LIN {X 0,Y 354.821,Z 300.916,A -85,B 0,C 180,E1 -13284.301,E2 -13284.301} C_VEL
LIN {X 0,Y 354.785,Z 300.918,A -85,B 0,C 180,E1 -13287.666,E2 -13287.666} C_VEL
LIN {X 0,Y 354.8,Z 300.915,A -85,B 0,C 180,E1 -13291.614,E2 -13291.614} C_VEL
LIN {X 0,Y 354.849,Z 300.908,A -85,B 0,C 180,E1 -13295.423,E2 -13295.423} C_VEL
LIN {X 0,Y 354.825,Z 300.912,A -85,B 0,C 180,E1 -13299.113,E2 -13299.113} C_VEL
LIN {X 0,Y 354.896,Z 300.903,A -85,B 0,C 180,E1 -13302.72,E2 -13302.72} C_VEL
LIN {X 0,Y 354.949,Z 300.895,A -85,B 0,C 180,E1 -13306.255,E2 -13306.255} C_VEL
LIN {X 0,Y 354.954,Z 300.896,A -85,B 0,C 180,E1 -13309.735,E2 -13309.735} C_VEL
LIN {X 0,Y 355.087,Z 300.878,A -85,B 0,C 180,E1 -13313.18,E2 -13313.18} C_VEL
LIN {X 0,Y 355.243,Z 300.859,A -85,B 0,C 180,E1 -13317.732,E2 -13317.732} C_VEL
LIN {X 0,Y 355.33,Z 300.85,A -85,B 0,C 180,E1 -13320,E2 -13320} C_VEL
LIN {X 0,Y 355.243,Z 300.859,A -85,B 0,C 180,E1 -13322.268,E2 -13322.268} C_VEL
LIN {X 0,Y 355.087,Z 300.878,A -85,B 0,C 180,E1 -13326.82,E2 -13326.82} C_VEL
LIN {X 0,Y 354.954,Z 300.896,A -85,B 0,C 180,E1 -13330.265,E2 -13330.265} C_VEL
LIN {X 0,Y 354.94,Z 300.899,A -85,B 0,C 180,E1 -13334.019,E2 -13334.019} C_VEL
LIN {X 0,Y 354.92,Z 300.901,A -85,B 0,C 180,E1 -13338.108,E2 -13338.108} C_VEL
LIN {X 0,Y 354.814,Z 300.913,A -85,B 0,C 180,E1 -13342.107,E2 -13342.107} C_VEL
LIN {X 0,Y 354.896,Z 300.904,A -85,B 0,C 180,E1 -13345.828,E2 -13345.828} C_VEL
LIN {X 0,Y 354.816,Z 300.917,A -85,B 0,C 180,E1 -13349.682,E2 -13349.682} C_VEL
LIN {X 0,Y 354.804,Z 300.923,A -85,B 0,C 180,E1 -13353.702,E2 -13353.702} C_VEL
LIN {X 0,Y 354.795,Z 300.924,A -85,B 0,C 180,E1 -13356.46,E2 -13356.46} C_VEL
LIN {X 0,Y 354.823,Z 300.917,A -85,B 0,C 180,E1 -13359.424,E2 -13359.424} C_VEL
LIN {X 0,Y 354.942,Z 301.94,A -85,B 0,C 180,E1 -13361.2,E2 -13361.2} C_VEL
LIN {X 0,Y 355.522,Z 305.414,A -85,B 0,C 180,E1 -13364.631,E2 -13364.631} C_VEL
LIN {X 0,Y 355.791,Z 308.9,A -85,B 0,C 180,E1 -13367.809,E2 -13367.809} C_VEL
LIN {X 0,Y 355.65,Z 312.374,A -85,B 0,C 180,E1 -13370.776,E2 -13370.776} C_VEL
LIN {X 0,Y 355.208,Z 316.65,A -85,B 0,C 180,E1 -13374.214,E2 -13374.214} C_VEL
LIN {X 0,Y 354.802,Z 321.128,A -85,B 0,C 180,E1 -13377.668,E2 -13377.668} C_VEL
LIN {X 0,Y 354.435,Z 325.194,A -85,B 0,C 180,E1 -13380.711,E2 -13380.711} C_VEL
LIN {X 0,Y 355.437,Z 328.521,A -85,B 0,C 180,E1 -13380.888,E2 -13380.888} C_VEL
LIN {X 0,Y 360.165,Z 342.303,A -85,B 0,C 180,E1 -13381.741,E2 -13381.741} C_VEL
LIN {X 0,Y 364.264,Z 357.145,A -85,B 0,C 180,E1 -13382.781,E2 -13382.781} C_VEL
LIN {X 0,Y 367.132,Z 370.992,A -85,B 0,C 180,E1 -13383.878,E2 -13383.878} C_VEL
LIN {X 0,Y 367.5,Z 375.118,A -85,B 0,C 180,E1 -13384.21,E2 -13384.21} C_VEL
LIN {X 0,Y 365.724,Z 389.395,A -85,B 0,C 180,E1 -13385.294,E2 -13385.294} C_VEL
LIN {X 0,Y 363.918,Z 402.392,A -85,B 0,C 180,E1 -13386.527,E2 -13386.527} C_VEL
LIN {X 0,Y 362.123,Z 414.391,A -85,B 0,C 180,E1 -13387.912,E2 -13387.912} C_VEL
LIN {X 0,Y 360.283,Z 425.503,A -85,B 0,C 180,E1 -13389.444,E2 -13389.444} C_VEL
LIN {X 0,Y 358.7,Z 435.728,A -85,B 0,C 180,E1 -13391.138,E2 -13391.138} C_VEL
LIN {X 0,Y 357.065,Z 445.72,A -85,B 0,C 180,E1 -13393.123,E2 -13393.123} C_VEL
LIN {X 0,Y 355.76,Z 454.016,A -85,B 0,C 180,E1 -13395.119,E2 -13395.119} C_VEL
LIN {X 0,Y 354.77,Z 461.81,A -85,B 0,C 180,E1 -13397.413,E2 -13397.413} C_VEL
LIN {X 0,Y 353.938,Z 468.009,A -85,B 0,C 180,E1 -13399.705,E2 -13399.705} C_VEL
LIN {X 0,Y 353.512,Z 472.803,A -85,B 0,C 180,E1 -13402,E2 -13402} C_VEL
LIN {X 0,Y 353.26,Z 476.314,A -85,B 0,C 180,E1 -13404.291,E2 -13404.291} C_VEL
LIN {X 0,Y 353.182,Z 478.624,A -85,B 0,C 180,E1 -13406.577,E2 -13406.577} C_VEL
LIN {X 0,Y 353.144,Z 479.785,A -85,B 0,C 180,E1 -13408.859,E2 -13408.859} C_VEL
LIN {X 0,Y 353.144,Z 479.783,A -85,B 0,C 180,E1 -13411.14,E2 -13411.14} C_VEL
LIN {X 0,Y 353.183,Z 478.613,A -85,B 0,C 180,E1 -13413.422,E2 -13413.422} C_VEL
LIN {X 0,Y 353.312,Z 475.97,A -85,B 0,C 180,E1 -13415.965,E2 -13415.965} C_VEL
LIN {X 0,Y 353.601,Z 471.718,A -85,B 0,C 180,E1 -13418.572,E2 -13418.572} C_VEL
LIN {X 0,Y 354.061,Z 466.558,A -85,B 0,C 180,E1 -13420.869,E2 -13420.869} C_VEL
LIN {X 0,Y 354.957,Z 459.959,A -85,B 0,C 180,E1 -13423.161,E2 -13423.161} C_VEL
LIN {X 0,Y 355.943,Z 452.851,A -85,B 0,C 180,E1 -13425.165,E2 -13425.165} C_VEL
LIN {X 0,Y 357.256,Z 444.313,A -85,B 0,C 180,E1 -13427.162,E2 -13427.162} C_VEL
LIN {X 0,Y 358.709,Z 435.666,A -85,B 0,C 180,E1 -13428.86,E2 -13428.86} C_VEL
LIN {X 0,Y 360.406,Z 425.069,A -85,B 0,C 180,E1 -13430.608,E2 -13430.608} C_VEL
LIN {X 0,Y 362.266,Z 413.241,A -85,B 0,C 180,E1 -13432.228,E2 -13432.228} C_VEL
LIN {X 0,Y 364.288,Z 399.662,A -85,B 0,C 180,E1 -13433.748,E2 -13433.748} C_VEL
LIN {X 0,Y 366.179,Z 386.045,A -85,B 0,C 180,E1 -13434.975,E2 -13434.975} C_VEL
LIN {X 0,Y 367.506,Z 374.442,A -85,B 0,C 180,E1 -13435.827,E2 -13435.827} C_VEL
LIN {X 0,Y 365.476,Z 363.038,A -85,B 0,C 180,E1 -13436.76,E2 -13436.76} C_VEL
LIN {X 0,Y 362.281,Z 349.698,A -85,B 0,C 180,E1 -13437.747,E2 -13437.747} C_VEL
LIN {X 0,Y 357.545,Z 334.313,A -85,B 0,C 180,E1 -13438.751,E2 -13438.751} C_VEL
LIN {X 0,Y 354.548,Z 326.07,A -85,B 0,C 180,E1 -13439.238,E2 -13439.238} C_VEL
LIN {X 0,Y 354.421,Z 325.198,A -85,B 0,C 180,E1 -13439.285,E2 -13439.285} C_VEL
LIN {X 0,Y 354.8,Z 321.14,A -85,B 0,C 180,E1 -13442.331,E2 -13442.331} C_VEL
LIN {X 0,Y 355.205,Z 316.687,A -85,B 0,C 180,E1 -13445.785,E2 -13445.785} C_VEL
LIN {X 0,Y 355.651,Z 312.432,A -85,B 0,C 180,E1 -13449.222,E2 -13449.222} C_VEL
LIN {X 0,Y 355.788,Z 308.925,A -85,B 0,C 180,E1 -13452.19,E2 -13452.19} C_VEL
LIN {X 0,Y 355.521,Z 305.416,A -85,B 0,C 180,E1 -13455.368,E2 -13455.368} C_VEL
LIN {X 0,Y 354.878,Z 301.531,A -85,B 0,C 180,E1 -13459.192,E2 -13459.192} C_VEL
LIN {X 0,Y 354.81,Z 300.916,A -85,B 0,C 180,E1 -13460.665,E2 -13460.665} C_VEL
LIN {X 0,Y 354.815,Z 300.917,A -85,B 0,C 180,E1 -13464.3,E2 -13464.3} C_VEL
LIN {X 0,Y 354.78,Z 300.924,A -85,B 0,C 180,E1 -13467.666,E2 -13467.666} C_VEL
LIN {X 0,Y 354.84,Z 300.914,A -85,B 0,C 180,E1 -13471.618,E2 -13471.618} C_VEL
LIN {X 0,Y 354.892,Z 300.905,A -85,B 0,C 180,E1 -13474.172,E2 -13474.172} C_VEL
LIN {X 0,Y 354.827,Z 300.911,A -85,B 0,C 180,E1 -13477.894,E2 -13477.894} C_VEL
LIN {X 0,Y 354.916,Z 300.9,A -85,B 0,C 180,E1 -13481.891,E2 -13481.891} C_VEL
LIN {X 0,Y 354.935,Z 300.897,A -85,B 0,C 180,E1 -13485.981,E2 -13485.981} C_VEL
LIN {X 0,Y 354.949,Z 300.896,A -85,B 0,C 180,E1 -13489.735,E2 -13489.735} C_VEL
LIN {X 0,Y 355.082,Z 300.879,A -85,B 0,C 180,E1 -13493.18,E2 -13493.18} C_VEL
LIN {X 0,Y 355.239,Z 300.855,A -85,B 0,C 180,E1 -13497.732,E2 -13497.732} C_VEL
LIN {X 0,Y 355.345,Z 300.849,A -85,B 0,C 180,E1 -13500,E2 -13500} C_VEL
LIN {X 0,Y 355.239,Z 300.859,A -85,B 0,C 180,E1 -13502.268,E2 -13502.268} C_VEL
LIN {X 0,Y 355.082,Z 300.879,A -85,B 0,C 180,E1 -13506.82,E2 -13506.82} C_VEL
LIN {X 0,Y 354.949,Z 300.897,A -85,B 0,C 180,E1 -13510.265,E2 -13510.265} C_VEL
LIN {X 0,Y 354.935,Z 300.897,A -85,B 0,C 180,E1 -13514.019,E2 -13514.019} C_VEL
LIN {X 0,Y 354.916,Z 300.898,A -85,B 0,C 180,E1 -13518.109,E2 -13518.109} C_VEL
LIN {X 0,Y 354.829,Z 300.911,A -85,B 0,C 180,E1 -13522.107,E2 -13522.107} C_VEL
LIN {X 0,Y 354.893,Z 300.904,A -85,B 0,C 180,E1 -13525.828,E2 -13525.828} C_VEL
LIN {X 0,Y 354.812,Z 300.91,A -85,B 0,C 180,E1 -13529.683,E2 -13529.683} C_VEL
LIN {X 0,Y 354.801,Z 300.913,A -85,B 0,C 180,E1 -13533.703,E2 -13533.703} C_VEL
LIN {X 0,Y 354.793,Z 300.915,A -85,B 0,C 180,E1 -13536.46,E2 -13536.46} C_VEL
LIN {X 0,Y 354.819,Z 300.914,A -85,B 0,C 180,E1 -13539.424,E2 -13539.424} C_VEL
LIN {X 0,Y 354.785,Z 300.92,A -85,B 0,C 180,E1 -13542.868,E2 -13542.868} C_VEL
LIN {X 0,Y 355.185,Z 303.837,A -85,B 0,C 180,E1 -13546.17,E2 -13546.17} C_VEL
LIN {X 0,Y 355.333,Z 306.315,A -85,B 0,C 180,E1 -13548.728,E2 -13548.728} C_VEL
LIN {X 0,Y 355.07,Z 309.877,A -85,B 0,C 180,E1 -13552.152,E2 -13552.152} C_VEL
LIN {X 0,Y 354.85,Z 312.922,A -85,B 0,C 180,E1 -13554.946,E2 -13554.946} C_VEL
LIN {X 0,Y 354.487,Z 317.485,A -85,B 0,C 180,E1 -13558.972,E2 -13558.972} C_VEL
LIN {X 0,Y 354.323,Z 319.729,A -85,B 0,C 180,E1 -13560.779,E2 -13560.779} C_VEL
LIN {X 0,Y 355.465,Z 323.077,A -85,B 0,C 180,E1 -13560.969,E2 -13560.969} C_VEL
LIN {X 0,Y 360.81,Z 337.991,A -85,B 0,C 180,E1 -13561.937,E2 -13561.937} C_VEL
LIN {X 0,Y 364.609,Z 351.156,A -85,B 0,C 180,E1 -13562.885,E2 -13562.885} C_VEL
LIN {X 0,Y 367.818,Z 365.813,A -85,B 0,C 180,E1 -13564.074,E2 -13564.074} C_VEL
LIN {X 0,Y 366.527,Z 379.062,A -85,B 0,C 180,E1 -13565.05,E2 -13565.05} C_VEL
LIN {X 0,Y 364.645,Z 392.749,A -85,B 0,C 180,E1 -13566.277,E2 -13566.277} C_VEL
LIN {X 0,Y 362.816,Z 405.219,A -85,B 0,C 180,E1 -13567.658,E2 -13567.658} C_VEL
LIN {X 0,Y 361.193,Z 415.771,A -85,B 0,C 180,E1 -13569.063,E2 -13569.063} C_VEL
LIN {X 0,Y 359.307,Z 427.192,A -85,B 0,C 180,E1 -13570.876,E2 -13570.876} C_VEL
LIN {X 0,Y 357.628,Z 437.465,A -85,B 0,C 180,E1 -13572.857,E2 -13572.857} C_VEL
LIN {X 0,Y 356.265,Z 445.996,A -85,B 0,C 180,E1 -13574.849,E2 -13574.849} C_VEL
LIN {X 0,Y 355.264,Z 453.095,A -85,B 0,C 180,E1 -13576.851,E2 -13576.851} C_VEL
LIN {X 0,Y 354.278,Z 459.684,A -85,B 0,C 180,E1 -13579.138,E2 -13579.138} C_VEL
LIN {X 0,Y 353.749,Z 464.834,A -85,B 0,C 180,E1 -13581.431,E2 -13581.431} C_VEL
LIN {X 0,Y 353.443,Z 468.827,A -85,B 0,C 180,E1 -13583.837,E2 -13583.837} C_VEL
LIN {X 0,Y 353.284,Z 470.71,A -85,B 0,C 180,E1 -13585.436,E2 -13585.436} C_VEL
LIN {X 0,Y 353.167,Z 472.459,A -85,B 0,C 180,E1 -13587.72,E2 -13587.72} C_VEL
LIN {X 0,Y 353.174,Z 473.069,A -85,B 0,C 180,E1 -13590,E2 -13590} C_VEL
LIN {X 0,Y 353.167,Z 472.503,A -85,B 0,C 180,E1 -13592.281,E2 -13592.281} C_VEL
LIN {X 0,Y 353.282,Z 470.812,A -85,B 0,C 180,E1 -13594.564,E2 -13594.564} C_VEL
LIN {X 0,Y 353.428,Z 467.96,A -85,B 0,C 180,E1 -13596.853,E2 -13596.853} C_VEL
LIN {X 0,Y 353.841,Z 463.877,A -85,B 0,C 180,E1 -13599.143,E2 -13599.143} C_VEL
LIN {X 0,Y 354.441,Z 458.466,A -85,B 0,C 180,E1 -13601.437,E2 -13601.437} C_VEL
LIN {X 0,Y 355.227,Z 453.413,A -85,B 0,C 180,E1 -13603.151,E2 -13603.151} C_VEL
LIN {X 0,Y 356.17,Z 446.386,A -85,B 0,C 180,E1 -13605.156,E2 -13605.156} C_VEL
LIN {X 0,Y 357.56,Z 437.93,A -85,B 0,C 180,E1 -13607.148,E2 -13607.148} C_VEL
LIN {X 0,Y 359.238,Z 427.749,A -85,B 0,C 180,E1 -13609.129,E2 -13609.129} C_VEL
LIN {X 0,Y 360.999,Z 417.043,A -85,B 0,C 180,E1 -13610.856,E2 -13610.856} C_VEL
LIN {X 0,Y 362.878,Z 404.837,A -85,B 0,C 180,E1 -13612.489,E2 -13612.489} C_VEL
LIN {X 0,Y 364.729,Z 392.289,A -85,B 0,C 180,E1 -13613.869,E2 -13613.869} C_VEL
LIN {X 0,Y 366.575,Z 379.12,A -85,B 0,C 180,E1 -13615.046,E2 -13615.046} C_VEL
LIN {X 0,Y 367.907,Z 366.961,A -85,B 0,C 180,E1 -13615.936,E2 -13615.936} C_VEL
LIN {X 0,Y 366.464,Z 359.08,A -85,B 0,C 180,E1 -13616.593,E2 -13616.593} C_VEL
LIN {X 0,Y 362.78,Z 344.309,A -85,B 0,C 180,E1 -13617.722,E2 -13617.722} C_VEL
LIN {X 0,Y 357.834,Z 329.329,A -85,B 0,C 180,E1 -13618.749,E2 -13618.749} C_VEL
LIN {X 0,Y 354.379,Z 320.072,A -85,B 0,C 180,E1 -13619.316,E2 -13619.316} C_VEL
LIN {X 0,Y 354.31,Z 319.565,A -85,B 0,C 180,E1 -13619.375,E2 -13619.375} C_VEL
LIN {X 0,Y 354.393,Z 318.435,A -85,B 0,C 180,E1 -13620.347,E2 -13620.347} C_VEL
LIN {X 0,Y 353.819,Z 317.434,A -85,B 0,C 180,E1 -13621.284,E2 -13621.284} C_VEL
LIN {X 0,Y 351.083,Z 316.043,A -85,B 0,C 180,E1 -13622.816,E2 -13622.816} C_VEL
LIN {X 0,Y 348.77,Z 314.97,A -85,B 0,C 180,E1 -13624.058,E2 -13624.058} C_VEL
LIN {X 0,Y 347.843,Z 314.059,A -85,B 0,C 180,E1 -13625.014,E2 -13625.014} C_VEL
LIN {X 0,Y 347.804,Z 313.72,A -85,B 0,C 180,E1 -13625.336,E2 -13625.336} C_VEL
LIN {X 0,Y 348.101,Z 310.13,A -85,B 0,C 180,E1 -13628.746,E2 -13628.746} C_VEL
LIN {X 0,Y 348.326,Z 307.061,A -85,B 0,C 180,E1 -13631.745,E2 -13631.745} C_VEL
LIN {X 0,Y 348.084,Z 304.026,A -85,B 0,C 180,E1 -13634.964,E2 -13634.964} C_VEL
LIN {X 0,Y 347.856,Z 302.5,A -85,B 0,C 180,E1 -13636.663,E2 -13636.663} C_VEL
LIN {X 0,Y 347.75,Z 301.794,A -85,B 0,C 180,E1 -13638.397,E2 -13638.397} C_VEL
LIN {X 0,Y 347.773,Z 301.793,A -85,B 0,C 180,E1 -13642.011,E2 -13642.011} C_VEL
LIN {X 0,Y 347.743,Z 301.797,A -85,B 0,C 180,E1 -13645.536,E2 -13645.536} C_VEL
LIN {X 0,Y 347.744,Z 301.796,A -85,B 0,C 180,E1 -13648.3,E2 -13648.3} C_VEL
LIN {X 0,Y 347.745,Z 301.794,A -85,B 0,C 180,E1 -13650.984,E2 -13650.984} C_VEL
LIN {X 0,Y 347.753,Z 301.791,A -85,B 0,C 180,E1 -13653.601,E2 -13653.601} C_VEL
LIN {X 0,Y 347.768,Z 301.791,A -85,B 0,C 180,E1 -13656.16,E2 -13656.16} C_VEL
LIN {X 0,Y 347.81,Z 301.787,A -85,B 0,C 180,E1 -13659.909,E2 -13659.909} C_VEL
LIN {X 0,Y 347.865,Z 301.779,A -85,B 0,C 180,E1 -13662.359,E2 -13662.359} C_VEL
LIN {X 0,Y 347.896,Z 301.776,A -85,B 0,C 180,E1 -13665.971,E2 -13665.971} C_VEL
LIN {X 0,Y 347.894,Z 301.776,A -85,B 0,C 180,E1 -13669.524,E2 -13669.524} C_VEL
LIN {X 0,Y 348.054,Z 301.755,A -85,B 0,C 180,E1 -13673.041,E2 -13673.041} C_VEL
LIN {X 0,Y 348.206,Z 301.735,A -85,B 0,C 180,E1 -13677.686,E2 -13677.686} C_VEL
LIN {X 0,Y 348.281,Z 301.728,A -85,B 0,C 180,E1 -13680,E2 -13680} C_VEL
LIN {X 0,Y 348.206,Z 301.736,A -85,B 0,C 180,E1 -13682.313,E2 -13682.313} C_VEL
LIN {X 0,Y 348.053,Z 301.754,A -85,B 0,C 180,E1 -13686.959,E2 -13686.959} C_VEL
LIN {X 0,Y 347.894,Z 301.777,A -85,B 0,C 180,E1 -13690.475,E2 -13690.475} C_VEL
LIN {X 0,Y 347.896,Z 301.776,A -85,B 0,C 180,E1 -13694.15,E2 -13694.15} C_VEL
LIN {X 0,Y 347.889,Z 301.778,A -85,B 0,C 180,E1 -13698.29,E2 -13698.29} C_VEL
LIN {X 0,Y 347.766,Z 301.793,A -85,B 0,C 180,E1 -13701.626,E2 -13701.626} C_VEL
LIN {X 0,Y 347.809,Z 301.785,A -85,B 0,C 180,E1 -13705.109,E2 -13705.109} C_VEL
LIN {X 0,Y 347.806,Z 301.789,A -85,B 0,C 180,E1 -13707.694,E2 -13707.694} C_VEL
LIN {X 0,Y 347.747,Z 301.799,A -85,B 0,C 180,E1 -13710.348,E2 -13710.348} C_VEL
LIN {X 0,Y 347.746,Z 301.802,A -85,B 0,C 180,E1 -13714.044,E2 -13714.044} C_VEL
LIN {X 0,Y 347.759,Z 301.8,A -85,B 0,C 180,E1 -13717.321,E2 -13717.321} C_VEL
LIN {X 0,Y 347.763,Z 301.892,A -85,B 0,C 180,E1 -13719.83,E2 -13719.83} C_VEL
LIN {X 0,Y 348.307,Z 305.371,A -85,B 0,C 180,E1 -13723.415,E2 -13723.415} C_VEL
LIN {X 0,Y 348.728,Z 308.572,A -85,B 0,C 180,E1 -13726.512,E2 -13726.512} C_VEL
LIN {X 0,Y 348.767,Z 310.573,A -85,B 0,C 180,E1 -13728.319,E2 -13728.319} C_VEL
LIN {X 0,Y 348.529,Z 314.056,A -85,B 0,C 180,E1 -13731.31,E2 -13731.31} C_VEL
LIN {X 0,Y 348.172,Z 317.564,A -85,B 0,C 180,E1 -13734.171,E2 -13734.171} C_VEL
LIN {X 0,Y 347.819,Z 321.054,A -85,B 0,C 180,E1 -13736.937,E2 -13736.937} C_VEL
LIN {X 0,Y 347.447,Z 325.114,A -85,B 0,C 180,E1 -13740.055,E2 -13740.055} C_VEL
LIN {X 0,Y 348.341,Z 328.241,A -85,B 0,C 180,E1 -13740.23,E2 -13740.23} C_VEL
LIN {X 0,Y 353.25,Z 342.107,A -85,B 0,C 180,E1 -13741.131,E2 -13741.131} C_VEL
LIN {X 0,Y 357.441,Z 357.227,A -85,B 0,C 180,E1 -13742.225,E2 -13742.225} C_VEL
LIN {X 0,Y 360.521,Z 372.091,A -85,B 0,C 180,E1 -13743.443,E2 -13743.443} C_VEL
LIN {X 0,Y 361.042,Z 375.23,A -85,B 0,C 180,E1 -13743.728,E2 -13743.728} C_VEL
LIN {X 0,Y 359.274,Z 389.33,A -85,B 0,C 180,E1 -13744.82,E2 -13744.82} C_VEL
LIN {X 0,Y 357.368,Z 402.326,A -85,B 0,C 180,E1 -13746.07,E2 -13746.07} C_VEL
LIN {X 0,Y 355.498,Z 414.325,A -85,B 0,C 180,E1 -13747.478,E2 -13747.478} C_VEL
LIN {X 0,Y 353.449,Z 426.184,A -85,B 0,C 180,E1 -13749.155,E2 -13749.155} C_VEL
LIN {X 0,Y 351.959,Z 435.661,A -85,B 0,C 180,E1 -13750.763,E2 -13750.763} C_VEL
LIN {X 0,Y 350.215,Z 445.652,A -85,B 0,C 180,E1 -13752.782,E2 -13752.782} C_VEL
LIN {X 0,Y 348.847,Z 453.948,A -85,B 0,C 180,E1 -13754.817,E2 -13754.817} C_VEL
LIN {X 0,Y 347.768,Z 461.742,A -85,B 0,C 180,E1 -13757.156,E2 -13757.156} C_VEL
LIN {X 0,Y 346.884,Z 467.94,A -85,B 0,C 180,E1 -13759.493,E2 -13759.493} C_VEL
LIN {X 0,Y 346.461,Z 472.734,A -85,B 0,C 180,E1 -13761.836,E2 -13761.836} C_VEL
LIN {X 0,Y 346.179,Z 476.246,A -85,B 0,C 180,E1 -13764.174,E2 -13764.174} C_VEL
LIN {X 0,Y 346.107,Z 478.556,A -85,B 0,C 180,E1 -13766.507,E2 -13766.507} C_VEL
LIN {X 0,Y 346.047,Z 479.716,A -85,B 0,C 180,E1 -13768.836,E2 -13768.836} C_VEL
LIN {X 0,Y 346.047,Z 479.714,A -85,B 0,C 180,E1 -13771.163,E2 -13771.163} C_VEL
LIN {X 0,Y 346.108,Z 478.544,A -85,B 0,C 180,E1 -13773.492,E2 -13773.492} C_VEL
LIN {X 0,Y 346.232,Z 476.081,A -85,B 0,C 180,E1 -13775.943,E2 -13775.943} C_VEL
LIN {X 0,Y 346.465,Z 472.716,A -85,B 0,C 180,E1 -13778.163,E2 -13778.163} C_VEL
LIN {X 0,Y 346.883,Z 467.917,A -85,B 0,C 180,E1 -13780.506,E2 -13780.506} C_VEL
LIN {X 0,Y 347.766,Z 461.703,A -85,B 0,C 180,E1 -13782.843,E2 -13782.843} C_VEL
LIN {X 0,Y 348.844,Z 453.898,A -85,B 0,C 180,E1 -13785.182,E2 -13785.182} C_VEL
LIN {X 0,Y 350.2,Z 445.597,A -85,B 0,C 180,E1 -13787.217,E2 -13787.217} C_VEL
LIN {X 0,Y 351.967,Z 435.595,A -85,B 0,C 180,E1 -13789.236,E2 -13789.236} C_VEL
LIN {X 0,Y 353.661,Z 425.363,A -85,B 0,C 180,E1 -13790.958,E2 -13790.958} C_VEL
LIN {X 0,Y 355.651,Z 413.169,A -85,B 0,C 180,E1 -13792.664,E2 -13792.664} C_VEL
LIN {X 0,Y 357.563,Z 400.926,A -85,B 0,C 180,E1 -13794.069,E2 -13794.069} C_VEL
LIN {X 0,Y 359.488,Z 387.6,A -85,B 0,C 180,E1 -13795.318,E2 -13795.318} C_VEL
LIN {X 0,Y 360.959,Z 375.6,A -85,B 0,C 180,E1 -13796.234,E2 -13796.234} C_VEL
LIN {X 0,Y 358.668,Z 362.956,A -85,B 0,C 180,E1 -13797.31,E2 -13797.31} C_VEL
LIN {X 0,Y 355.534,Z 349.991,A -85,B 0,C 180,E1 -13798.302,E2 -13798.302} C_VEL
LIN {X 0,Y 350.925,Z 335.076,A -85,B 0,C 180,E1 -13799.316,E2 -13799.316} C_VEL
LIN {X 0,Y 347.532,Z 325.872,A -85,B 0,C 180,E1 -13799.89,E2 -13799.89} C_VEL
LIN {X 0,Y 347.428,Z 325.084,A -85,B 0,C 180,E1 -13799.966,E2 -13799.966} C_VEL
LIN {X 0,Y 347.817,Z 321.068,A -85,B 0,C 180,E1 -13803.062,E2 -13803.062} C_VEL
LIN {X 0,Y 348.222,Z 317.169,A -85,B 0,C 180,E1 -13806.167,E2 -13806.167} C_VEL
LIN {X 0,Y 348.528,Z 314.105,A -85,B 0,C 180,E1 -13808.689,E2 -13808.689} C_VEL
LIN {X 0,Y 348.764,Z 310.487,A -85,B 0,C 180,E1 -13811.79,E2 -13811.79} C_VEL
LIN {X 0,Y 348.59,Z 307.102,A -85,B 0,C 180,E1 -13814.88,E2 -13814.88} C_VEL
LIN {X 0,Y 348.021,Z 303.604,A -85,B 0,C 180,E1 -13818.345,E2 -13818.345} C_VEL
LIN {X 0,Y 347.756,Z 301.857,A -85,B 0,C 180,E1 -13820.17,E2 -13820.17} C_VEL
LIN {X 0,Y 347.764,Z 301.795,A -85,B 0,C 180,E1 -13823.934,E2 -13823.934} C_VEL
LIN {X 0,Y 347.726,Z 301.802,A -85,B 0,C 180,E1 -13826.927,E2 -13826.927} C_VEL
LIN {X 0,Y 347.772,Z 301.795,A -85,B 0,C 180,E1 -13830.987,E2 -13830.987} C_VEL
LIN {X 0,Y 347.824,Z 301.787,A -85,B 0,C 180,E1 -13833.607,E2 -13833.607} C_VEL
LIN {X 0,Y 347.781,Z 301.789,A -85,B 0,C 180,E1 -13836.162,E2 -13836.162} C_VEL
LIN {X 0,Y 347.81,Z 301.787,A -85,B 0,C 180,E1 -13839.909,E2 -13839.909} C_VEL
LIN {X 0,Y 347.859,Z 301.778,A -85,B 0,C 180,E1 -13842.359,E2 -13842.359} C_VEL
LIN {X 0,Y 347.89,Z 301.774,A -85,B 0,C 180,E1 -13845.971,E2 -13845.971} C_VEL
LIN {X 0,Y 347.889,Z 301.777,A -85,B 0,C 180,E1 -13849.525,E2 -13849.525} C_VEL
LIN {X 0,Y 348.048,Z 301.755,A -85,B 0,C 180,E1 -13853.041,E2 -13853.041} C_VEL
LIN {X 0,Y 348.201,Z 301.731,A -85,B 0,C 180,E1 -13857.687,E2 -13857.687} C_VEL
LIN {X 0,Y 348.296,Z 301.726,A -85,B 0,C 180,E1 -13860,E2 -13860} C_VEL
LIN {X 0,Y 348.201,Z 301.736,A -85,B 0,C 180,E1 -13862.314,E2 -13862.314} C_VEL
LIN {X 0,Y 348.049,Z 301.756,A -85,B 0,C 180,E1 -13866.959,E2 -13866.959} C_VEL
LIN {X 0,Y 347.889,Z 301.777,A -85,B 0,C 180,E1 -13870.476,E2 -13870.476} C_VEL
LIN {X 0,Y 347.892,Z 301.773,A -85,B 0,C 180,E1 -13874.15,E2 -13874.15} C_VEL
LIN {X 0,Y 347.885,Z 301.775,A -85,B 0,C 180,E1 -13878.291,E2 -13878.291} C_VEL
LIN {X 0,Y 347.783,Z 301.79,A -85,B 0,C 180,E1 -13881.636,E2 -13881.636} C_VEL
LIN {X 0,Y 347.806,Z 301.785,A -85,B 0,C 180,E1 -13885.109,E2 -13885.109} C_VEL
LIN {X 0,Y 347.802,Z 301.785,A -85,B 0,C 180,E1 -13887.695,E2 -13887.695} C_VEL
LIN {X 0,Y 347.743,Z 301.791,A -85,B 0,C 180,E1 -13890.349,E2 -13890.349} C_VEL
LIN {X 0,Y 347.743,Z 301.792,A -85,B 0,C 180,E1 -13894.045,E2 -13894.045} C_VEL
LIN {X 0,Y 347.757,Z 301.792,A -85,B 0,C 180,E1 -13897.322,E2 -13897.322} C_VEL
LIN {X 0,Y 347.728,Z 301.798,A -85,B 0,C 180,E1 -13900.298,E2 -13900.298} C_VEL
LIN {X 0,Y 347.746,Z 301.796,A -85,B 0,C 180,E1 -13901.831,E2 -13901.831} C_VEL
LIN {X 0,Y 347.821,Z 302.435,A -85,B 0,C 180,E1 -13903.393,E2 -13903.393} C_VEL
LIN {X 0,Y 348.228,Z 305.411,A -85,B 0,C 180,E1 -13906.672,E2 -13906.672} C_VEL
LIN {X 0,Y 348.321,Z 306.95,A -85,B 0,C 180,E1 -13908.292,E2 -13908.292} C_VEL
LIN {X 0,Y 348.093,Z 309.944,A -85,B 0,C 180,E1 -13911.254,E2 -13911.254} C_VEL
LIN {X 0,Y 347.897,Z 312.987,A -85,B 0,C 180,E1 -13914.139,E2 -13914.139} C_VEL
LIN {X 0,Y 347.494,Z 317.552,A -85,B 0,C 180,E1 -13918.276,E2 -13918.276} C_VEL
LIN {X 0,Y 347.332,Z 319.742,A -85,B 0,C 180,E1 -13920.129,E2 -13920.129} C_VEL
LIN {X 0,Y 348.349,Z 322.945,A -85,B 0,C 180,E1 -13920.311,E2 -13920.311} C_VEL
LIN {X 0,Y 353.631,Z 337.175,A -85,B 0,C 180,E1 -13921.275,E2 -13921.275} C_VEL
LIN {X 0,Y 357.71,Z 350.899,A -85,B 0,C 180,E1 -13922.299,E2 -13922.299} C_VEL
LIN {X 0,Y 361.083,Z 365.858,A -85,B 0,C 180,E1 -13923.551,E2 -13923.551} C_VEL
LIN {X 0,Y 361.215,Z 369.406,A -85,B 0,C 180,E1 -13923.839,E2 -13923.839} C_VEL
LIN {X 0,Y 359.399,Z 383.979,A -85,B 0,C 180,E1 -13924.985,E2 -13924.985} C_VEL
LIN {X 0,Y 357.566,Z 396.776,A -85,B 0,C 180,E1 -13926.239,E2 -13926.239} C_VEL
LIN {X 0,Y 355.518,Z 409.671,A -85,B 0,C 180,E1 -13927.787,E2 -13927.787} C_VEL
LIN {X 0,Y 353.783,Z 420.451,A -85,B 0,C 180,E1 -13929.354,E2 -13929.354} C_VEL
LIN {X 0,Y 352.052,Z 430.42,A -85,B 0,C 180,E1 -13931.072,E2 -13931.072} C_VEL
LIN {X 0,Y 350.362,Z 440.157,A -85,B 0,C 180,E1 -13933.091,E2 -13933.091} C_VEL
LIN {X 0,Y 348.952,Z 448.476,A -85,B 0,C 180,E1 -13935.181,E2 -13935.181} C_VEL
LIN {X 0,Y 348.035,Z 454.97,A -85,B 0,C 180,E1 -13937.167,E2 -13937.167} C_VEL
LIN {X 0,Y 347.12,Z 461.174,A -85,B 0,C 180,E1 -13939.502,E2 -13939.502} C_VEL
LIN {X 0,Y 346.561,Z 465.964,A -85,B 0,C 180,E1 -13941.84,E2 -13941.84} C_VEL
LIN {X 0,Y 346.289,Z 469.474,A -85,B 0,C 180,E1 -13944.176,E2 -13944.176} C_VEL
LIN {X 0,Y 346.142,Z 471.795,A -85,B 0,C 180,E1 -13946.508,E2 -13946.508} C_VEL
LIN {X 0,Y 346.058,Z 472.98,A -85,B 0,C 180,E1 -13948.837,E2 -13948.837} C_VEL
LIN {X 0,Y 346.059,Z 472.995,A -85,B 0,C 180,E1 -13951.164,E2 -13951.164} C_VEL
LIN {X 0,Y 346.142,Z 471.868,A -85,B 0,C 180,E1 -13953.493,E2 -13953.493} C_VEL
LIN {X 0,Y 346.325,Z 469.278,A -85,B 0,C 180,E1 -13956.087,E2 -13956.087} C_VEL
LIN {X 0,Y 346.685,Z 465.084,A -85,B 0,C 180,E1 -13958.745,E2 -13958.745} C_VEL
LIN {X 0,Y 347.255,Z 459.996,A -85,B 0,C 180,E1 -13961.085,E2 -13961.085} C_VEL
LIN {X 0,Y 348.259,Z 453.481,A -85,B 0,C 180,E1 -13963.419,E2 -13963.419} C_VEL
LIN {X 0,Y 349.454,Z 445.34,A -85,B 0,C 180,E1 -13965.754,E2 -13965.754} C_VEL
LIN {X 0,Y 350.964,Z 436.646,A -85,B 0,C 180,E1 -13967.781,E2 -13967.781} C_VEL
LIN {X 0,Y 352.509,Z 427.815,A -85,B 0,C 180,E1 -13969.509,E2 -13969.509} C_VEL
LIN {X 0,Y 354.224,Z 417.771,A -85,B 0,C 180,E1 -13971.171,E2 -13971.171} C_VEL
LIN {X 0,Y 356.12,Z 406.073,A -85,B 0,C 180,E1 -13972.787,E2 -13972.787} C_VEL
LIN {X 0,Y 358.022,Z 393.761,A -85,B 0,C 180,E1 -13974.191,E2 -13974.191} C_VEL
LIN {X 0,Y 359.963,Z 380.301,A -85,B 0,C 180,E1 -13975.438,E2 -13975.438} C_VEL
LIN {X 0,Y 361.374,Z 367.72,A -85,B 0,C 180,E1 -13976.386,E2 -13976.386} C_VEL
LIN {X 0,Y 358.6,Z 354.586,A -85,B 0,C 180,E1 -13977.508,E2 -13977.508} C_VEL
LIN {X 0,Y 354.962,Z 341.471,A -85,B 0,C 180,E1 -13978.524,E2 -13978.524} C_VEL
LIN {X 0,Y 350.154,Z 327.426,A -85,B 0,C 180,E1 -13979.506,E2 -13979.506} C_VEL
LIN {X 0,Y 347.498,Z 320.697,A -85,B 0,C 180,E1 -13979.941,E2 -13979.941} C_VEL
LIN {X 0,Y 347.309,Z 319.651,A -85,B 0,C 180,E1 -13980.006,E2 -13980.006} C_VEL
LIN {X 0,Y 347.596,Z 316.174,A -85,B 0,C 180,E1 -13983.087,E2 -13983.087} C_VEL
LIN {X 0,Y 347.804,Z 313.72,A -85,B 0,C 180,E1 -13985.336,E2 -13985.336} C_VEL
LIN {X 0,Y 347.272,Z 312.789,A -85,B 0,C 180,E1 -13986.292,E2 -13986.292} C_VEL
LIN {X 0,Y 344.604,Z 311.543,A -85,B 0,C 180,E1 -13987.858,E2 -13987.858} C_VEL
LIN {X 0,Y 342.289,Z 310.57,A -85,B 0,C 180,E1 -13989.126,E2 -13989.126} C_VEL
LIN {X 0,Y 341.297,Z 309.734,A -85,B 0,C 180,E1 -13990.103,E2 -13990.103} C_VEL
LIN {X 0,Y 341.221,Z 309.422,A -85,B 0,C 180,E1 -13990.433,E2 -13990.433} C_VEL
LIN {X 0,Y 341.242,Z 307.135,A -85,B 0,C 180,E1 -13992.816,E2 -13992.816} C_VEL
LIN {X 0,Y 340.881,Z 304.078,A -85,B 0,C 180,E1 -13996.187,E2 -13996.187} C_VEL
LIN {X 0,Y 340.694,Z 302.673,A -85,B 0,C 180,E1 -13997.955,E2 -13997.955} C_VEL
LIN {X 0,Y 340.732,Z 302.671,A -85,B 0,C 180,E1 -14001.772,E2 -14001.772} C_VEL
LIN {X 0,Y 340.722,Z 302.671,A -85,B 0,C 180,E1 -14005.595,E2 -14005.595} C_VEL
LIN {X 0,Y 340.693,Z 302.674,A -85,B 0,C 180,E1 -14008.955,E2 -14008.955} C_VEL
LIN {X 0,Y 340.721,Z 302.667,A -85,B 0,C 180,E1 -14013.013,E2 -14013.013} C_VEL
LIN {X 0,Y 340.741,Z 302.666,A -85,B 0,C 180,E1 -14015.637,E2 -14015.637} C_VEL
LIN {X 0,Y 340.735,Z 302.667,A -85,B 0,C 180,E1 -14019.473,E2 -14019.473} C_VEL
LIN {X 0,Y 340.856,Z 302.653,A -85,B 0,C 180,E1 -14021.984,E2 -14021.984} C_VEL
LIN {X 0,Y 340.868,Z 302.65,A -85,B 0,C 180,E1 -14025.705,E2 -14025.705} C_VEL
LIN {X 0,Y 340.846,Z 302.655,A -85,B 0,C 180,E1 -14029.305,E2 -14029.305} C_VEL
LIN {X 0,Y 341.001,Z 302.634,A -85,B 0,C 180,E1 -14032.897,E2 -14032.897} C_VEL
LIN {X 0,Y 341.167,Z 302.612,A -85,B 0,C 180,E1 -14037.639,E2 -14037.639} C_VEL
LIN {X 0,Y 341.233,Z 302.606,A -85,B 0,C 180,E1 -14040,E2 -14040} C_VEL
LIN {X 0,Y 341.167,Z 302.613,A -85,B 0,C 180,E1 -14042.361,E2 -14042.361} C_VEL
LIN {X 0,Y 341,Z 302.633,A -85,B 0,C 180,E1 -14047.103,E2 -14047.103} C_VEL
LIN {X 0,Y 340.846,Z 302.654,A -85,B 0,C 180,E1 -14050.694,E2 -14050.694} C_VEL
LIN {X 0,Y 340.861,Z 302.652,A -85,B 0,C 180,E1 -14054.325,E2 -14054.325} C_VEL
LIN {X 0,Y 340.835,Z 302.657,A -85,B 0,C 180,E1 -14058.466,E2 -14058.466} C_VEL
LIN {X 0,Y 340.716,Z 302.67,A -85,B 0,C 180,E1 -14061.842,E2 -14061.842} C_VEL
LIN {X 0,Y 340.769,Z 302.663,A -85,B 0,C 180,E1 -14065.664,E2 -14065.664} C_VEL
LIN {X 0,Y 340.726,Z 302.671,A -85,B 0,C 180,E1 -14068.321,E2 -14068.321} C_VEL
LIN {X 0,Y 340.696,Z 302.678,A -85,B 0,C 180,E1 -14071.045,E2 -14071.045} C_VEL
LIN {X 0,Y 340.716,Z 302.679,A -85,B 0,C 180,E1 -14075.279,E2 -14075.279} C_VEL
LIN {X 0,Y 340.707,Z 302.678,A -85,B 0,C 180,E1 -14078.386,E2 -14078.386} C_VEL
LIN {X 0,Y 340.776,Z 303.075,A -85,B 0,C 180,E1 -14079.742,E2 -14079.742} C_VEL
LIN {X 0,Y 341.191,Z 305.986,A -85,B 0,C 180,E1 -14082.824,E2 -14082.824} C_VEL
LIN {X 0,Y 341.625,Z 308.791,A -85,B 0,C 180,E1 -14085.617,E2 -14085.617} C_VEL
LIN {X 0,Y 341.735,Z 311.059,A -85,B 0,C 180,E1 -14087.762,E2 -14087.762} C_VEL
LIN {X 0,Y 341.6,Z 314.005,A -85,B 0,C 180,E1 -14090.373,E2 -14090.373} C_VEL
LIN {X 0,Y 341.244,Z 317.615,A -85,B 0,C 180,E1 -14093.438,E2 -14093.438} C_VEL
LIN {X 0,Y 340.866,Z 320.988,A -85,B 0,C 180,E1 -14096.173,E2 -14096.173} C_VEL
LIN {X 0,Y 340.467,Z 325.031,A -85,B 0,C 180,E1 -14099.367,E2 -14099.367} C_VEL
LIN {X 0,Y 341.485,Z 328.364,A -85,B 0,C 180,E1 -14099.575,E2 -14099.575} C_VEL
LIN {X 0,Y 346.646,Z 342.896,A -85,B 0,C 180,E1 -14100.565,E2 -14100.565} C_VEL
LIN {X 0,Y 350.748,Z 357.451,A -85,B 0,C 180,E1 -14101.665,E2 -14101.665} C_VEL
LIN {X 0,Y 353.699,Z 371.787,A -85,B 0,C 180,E1 -14102.872,E2 -14102.872} C_VEL
LIN {X 0,Y 354.505,Z 376.519,A -85,B 0,C 180,E1 -14103.313,E2 -14103.313} C_VEL
LIN {X 0,Y 352.617,Z 390.848,A -85,B 0,C 180,E1 -14104.468,E2 -14104.468} C_VEL
LIN {X 0,Y 350.677,Z 403.552,A -85,B 0,C 180,E1 -14105.742,E2 -14105.742} C_VEL
LIN {X 0,Y 348.536,Z 416.4,A -85,B 0,C 180,E1 -14107.316,E2 -14107.316} C_VEL
LIN {X 0,Y 346.437,Z 428.29,A -85,B 0,C 180,E1 -14109.092,E2 -14109.092} C_VEL
LIN {X 0,Y 344.581,Z 438.593,A -85,B 0,C 180,E1 -14110.954,E2 -14110.954} C_VEL
LIN {X 0,Y 342.947,Z 448.073,A -85,B 0,C 180,E1 -14113.021,E2 -14113.021} C_VEL
LIN {X 0,Y 341.594,Z 455.858,A -85,B 0,C 180,E1 -14115.063,E2 -14115.063} C_VEL
LIN {X 0,Y 340.539,Z 463.343,A -85,B 0,C 180,E1 -14117.485,E2 -14117.485} C_VEL
LIN {X 0,Y 339.715,Z 469.189,A -85,B 0,C 180,E1 -14119.872,E2 -14119.872} C_VEL
LIN {X 0,Y 339.394,Z 472.666,A -85,B 0,C 180,E1 -14121.665,E2 -14121.665} C_VEL
LIN {X 0,Y 339.086,Z 476.345,A -85,B 0,C 180,E1 -14124.189,E2 -14124.189} C_VEL
LIN {X 0,Y 339.032,Z 478.487,A -85,B 0,C 180,E1 -14126.434,E2 -14126.434} C_VEL
LIN {X 0,Y 338.953,Z 479.647,A -85,B 0,C 180,E1 -14128.811,E2 -14128.811} C_VEL
LIN {X 0,Y 338.953,Z 479.645,A -85,B 0,C 180,E1 -14131.188,E2 -14131.188} C_VEL
LIN {X 0,Y 339.034,Z 478.475,A -85,B 0,C 180,E1 -14133.565,E2 -14133.565} C_VEL
LIN {X 0,Y 339.131,Z 476.158,A -85,B 0,C 180,E1 -14135.947,E2 -14135.947} C_VEL
LIN {X 0,Y 339.396,Z 472.646,A -85,B 0,C 180,E1 -14138.334,E2 -14138.334} C_VEL
LIN {X 0,Y 339.842,Z 467.846,A -85,B 0,C 180,E1 -14140.726,E2 -14140.726} C_VEL
LIN {X 0,Y 340.762,Z 461.632,A -85,B 0,C 180,E1 -14143.112,E2 -14143.112} C_VEL
LIN {X 0,Y 341.937,Z 453.827,A -85,B 0,C 180,E1 -14145.497,E2 -14145.497} C_VEL
LIN {X 0,Y 343.375,Z 445.525,A -85,B 0,C 180,E1 -14147.571,E2 -14147.571} C_VEL
LIN {X 0,Y 345.237,Z 435.523,A -85,B 0,C 180,E1 -14149.626,E2 -14149.626} C_VEL
LIN {X 0,Y 346.983,Z 425.291,A -85,B 0,C 180,E1 -14151.381,E2 -14151.381} C_VEL
LIN {X 0,Y 349.087,Z 413.096,A -85,B 0,C 180,E1 -14153.114,E2 -14153.114} C_VEL
LIN {X 0,Y 351.08,Z 400.854,A -85,B 0,C 180,E1 -14154.542,E2 -14154.542} C_VEL
LIN {X 0,Y 353.073,Z 387.527,A -85,B 0,C 180,E1 -14155.812,E2 -14155.812} C_VEL
LIN {X 0,Y 354.428,Z 376.703,A -85,B 0,C 180,E1 -14156.662,E2 -14156.662} C_VEL
LIN {X 0,Y 352.158,Z 364.05,A -85,B 0,C 180,E1 -14157.786,E2 -14157.786} C_VEL
LIN {X 0,Y 348.585,Z 349.526,A -85,B 0,C 180,E1 -14158.938,E2 -14158.938} C_VEL
LIN {X 0,Y 343.92,Z 334.931,A -85,B 0,C 180,E1 -14159.975,E2 -14159.975} C_VEL
LIN {X 0,Y 340.575,Z 325.969,A -85,B 0,C 180,E1 -14160.561,E2 -14160.561} C_VEL
LIN {X 0,Y 340.443,Z 324.998,A -85,B 0,C 180,E1 -14160.656,E2 -14160.656} C_VEL
LIN {X 0,Y 340.862,Z 320.998,A -85,B 0,C 180,E1 -14163.826,E2 -14163.826} C_VEL
LIN {X 0,Y 341.253,Z 317.512,A -85,B 0,C 180,E1 -14166.672,E2 -14166.672} C_VEL
LIN {X 0,Y 341.598,Z 314.04,A -85,B 0,C 180,E1 -14169.626,E2 -14169.626} C_VEL
LIN {X 0,Y 341.719,Z 310.545,A -85,B 0,C 180,E1 -14172.741,E2 -14172.741} C_VEL
LIN {X 0,Y 341.488,Z 307.54,A -85,B 0,C 180,E1 -14175.594,E2 -14175.594} C_VEL
LIN {X 0,Y 340.97,Z 304.475,A -85,B 0,C 180,E1 -14178.733,E2 -14178.733} C_VEL
LIN {X 0,Y 340.77,Z 303.046,A -85,B 0,C 180,E1 -14180.257,E2 -14180.257} C_VEL
LIN {X 0,Y 340.727,Z 302.671,A -85,B 0,C 180,E1 -14181.772,E2 -14181.772} C_VEL
LIN {X 0,Y 340.717,Z 302.675,A -85,B 0,C 180,E1 -14185.595,E2 -14185.595} C_VEL
LIN {X 0,Y 340.691,Z 302.679,A -85,B 0,C 180,E1 -14188.955,E2 -14188.955} C_VEL
LIN {X 0,Y 340.796,Z 302.662,A -85,B 0,C 180,E1 -14193.019,E2 -14193.019} C_VEL
LIN {X 0,Y 340.749,Z 302.667,A -85,B 0,C 180,E1 -14195.638,E2 -14195.638} C_VEL
LIN {X 0,Y 340.748,Z 302.665,A -85,B 0,C 180,E1 -14199.474,E2 -14199.474} C_VEL
LIN {X 0,Y 340.851,Z 302.652,A -85,B 0,C 180,E1 -14201.984,E2 -14201.984} C_VEL
LIN {X 0,Y 340.862,Z 302.648,A -85,B 0,C 180,E1 -14205.705,E2 -14205.705} C_VEL
LIN {X 0,Y 340.841,Z 302.656,A -85,B 0,C 180,E1 -14209.305,E2 -14209.305} C_VEL
LIN {X 0,Y 340.995,Z 302.634,A -85,B 0,C 180,E1 -14212.897,E2 -14212.897} C_VEL
LIN {X 0,Y 341.163,Z 302.608,A -85,B 0,C 180,E1 -14217.639,E2 -14217.639} C_VEL
LIN {X 0,Y 341.248,Z 302.604,A -85,B 0,C 180,E1 -14220,E2 -14220} C_VEL
LIN {X 0,Y 341.163,Z 302.612,A -85,B 0,C 180,E1 -14222.361,E2 -14222.361} C_VEL
LIN {X 0,Y 340.995,Z 302.634,A -85,B 0,C 180,E1 -14227.104,E2 -14227.104} C_VEL
LIN {X 0,Y 340.841,Z 302.654,A -85,B 0,C 180,E1 -14230.695,E2 -14230.695} C_VEL
LIN {X 0,Y 340.856,Z 302.649,A -85,B 0,C 180,E1 -14234.325,E2 -14234.325} C_VEL
LIN {X 0,Y 340.831,Z 302.655,A -85,B 0,C 180,E1 -14238.467,E2 -14238.467} C_VEL
LIN {X 0,Y 340.747,Z 302.665,A -85,B 0,C 180,E1 -14241.857,E2 -14241.857} C_VEL
LIN {X 0,Y 340.766,Z 302.663,A -85,B 0,C 180,E1 -14245.665,E2 -14245.665} C_VEL
LIN {X 0,Y 340.722,Z 302.665,A -85,B 0,C 180,E1 -14248.321,E2 -14248.321} C_VEL
LIN {X 0,Y 340.692,Z 302.668,A -85,B 0,C 180,E1 -14251.045,E2 -14251.045} C_VEL
LIN {X 0,Y 340.713,Z 302.669,A -85,B 0,C 180,E1 -14255.28,E2 -14255.28} C_VEL
LIN {X 0,Y 340.705,Z 302.672,A -85,B 0,C 180,E1 -14258.387,E2 -14258.387} C_VEL
LIN {X 0,Y 340.686,Z 302.675,A -85,B 0,C 180,E1 -14262.045,E2 -14262.045} C_VEL
LIN {X 0,Y 340.946,Z 304.55,A -85,B 0,C 180,E1 -14264.495,E2 -14264.495} C_VEL
LIN {X 0,Y 341.255,Z 307.609,A -85,B 0,C 180,E1 -14267.851,E2 -14267.851} C_VEL
LIN {X 0,Y 341.16,Z 310.01,A -85,B 0,C 180,E1 -14270.313,E2 -14270.313} C_VEL
LIN {X 0,Y 340.886,Z 313.309,A -85,B 0,C 180,E1 -14273.52,E2 -14273.52} C_VEL
LIN {X 0,Y 340.618,Z 316.103,A -85,B 0,C 180,E1 -14276.146,E2 -14276.146} C_VEL
LIN {X 0,Y 340.326,Z 319.713,A -85,B 0,C 180,E1 -14279.428,E2 -14279.428} C_VEL
LIN {X 0,Y 341.365,Z 323.019,A -85,B 0,C 180,E1 -14279.639,E2 -14279.639} C_VEL
LIN {X 0,Y 346.717,Z 337.281,A -85,B 0,C 180,E1 -14280.647,E2 -14280.647} C_VEL
LIN {X 0,Y 351.035,Z 351.457,A -85,B 0,C 180,E1 -14281.753,E2 -14281.753} C_VEL
LIN {X 0,Y 354.207,Z 365.574,A -85,B 0,C 180,E1 -14282.969,E2 -14282.969} C_VEL
LIN {X 0,Y 354.839,Z 369.482,A -85,B 0,C 180,E1 -14283.332,E2 -14283.332} C_VEL
LIN {X 0,Y 352.975,Z 384.053,A -85,B 0,C 180,E1 -14284.497,E2 -14284.497} C_VEL
LIN {X 0,Y 351.025,Z 396.85,A -85,B 0,C 180,E1 -14285.769,E2 -14285.769} C_VEL
LIN {X 0,Y 348.93,Z 409.744,A -85,B 0,C 180,E1 -14287.344,E2 -14287.344} C_VEL
LIN {X 0,Y 347.119,Z 420.524,A -85,B 0,C 180,E1 -14288.939,E2 -14288.939} C_VEL
LIN {X 0,Y 345.276,Z 430.492,A -85,B 0,C 180,E1 -14290.686,E2 -14290.686} C_VEL
LIN {X 0,Y 343.527,Z 440.229,A -85,B 0,C 180,E1 -14292.744,E2 -14292.744} C_VEL
LIN {X 0,Y 341.945,Z 449.026,A -85,B 0,C 180,E1 -14295.015,E2 -14295.015} C_VEL
LIN {X 0,Y 340.797,Z 456.721,A -85,B 0,C 180,E1 -14297.495,E2 -14297.495} C_VEL
LIN {X 0,Y 339.92,Z 462.571,A -85,B 0,C 180,E1 -14299.879,E2 -14299.879} C_VEL
LIN {X 0,Y 339.519,Z 466.035,A -85,B 0,C 180,E1 -14301.669,E2 -14301.669} C_VEL
LIN {X 0,Y 339.209,Z 469.544,A -85,B 0,C 180,E1 -14304.054,E2 -14304.054} C_VEL
LIN {X 0,Y 339.069,Z 471.864,A -85,B 0,C 180,E1 -14306.435,E2 -14306.435} C_VEL
LIN {X 0,Y 338.964,Z 473.049,A -85,B 0,C 180,E1 -14308.812,E2 -14308.812} C_VEL
LIN {X 0,Y 338.965,Z 473.064,A -85,B 0,C 180,E1 -14311.188,E2 -14311.188} C_VEL
LIN {X 0,Y 339.068,Z 471.937,A -85,B 0,C 180,E1 -14313.565,E2 -14313.565} C_VEL
LIN {X 0,Y 339.245,Z 469.526,A -85,B 0,C 180,E1 -14316.067,E2 -14316.067} C_VEL
LIN {X 0,Y 339.517,Z 466.214,A -85,B 0,C 180,E1 -14318.332,E2 -14318.332} C_VEL
LIN {X 0,Y 340.065,Z 461.482,A -85,B 0,C 180,E1 -14320.72,E2 -14320.72} C_VEL
LIN {X 0,Y 341.04,Z 455.351,A -85,B 0,C 180,E1 -14323.102,E2 -14323.102} C_VEL
LIN {X 0,Y 342.207,Z 447.634,A -85,B 0,C 180,E1 -14325.485,E2 -14325.485} C_VEL
LIN {X 0,Y 343.679,Z 439.407,A -85,B 0,C 180,E1 -14327.556,E2 -14327.556} C_VEL
LIN {X 0,Y 345.468,Z 429.498,A -85,B 0,C 180,E1 -14329.613,E2 -14329.613} C_VEL
LIN {X 0,Y 347.447,Z 418.532,A -85,B 0,C 180,E1 -14331.492,E2 -14331.492} C_VEL
LIN {X 0,Y 349.556,Z 406.139,A -85,B 0,C 180,E1 -14333.239,E2 -14333.239} C_VEL
LIN {X 0,Y 351.519,Z 393.826,A -85,B 0,C 180,E1 -14334.668,E2 -14334.668} C_VEL
LIN {X 0,Y 353.575,Z 380.365,A -85,B 0,C 180,E1 -14335.931,E2 -14335.931} C_VEL
LIN {X 0,Y 354.877,Z 369.502,A -85,B 0,C 180,E1 -14336.77,E2 -14336.77} C_VEL
LIN {X 0,Y 352.102,Z 355.859,A -85,B 0,C 180,E1 -14337.985,E2 -14337.985} C_VEL
LIN {X 0,Y 348.435,Z 342.561,A -85,B 0,C 180,E1 -14339.062,E2 -14339.062} C_VEL
LIN {X 0,Y 343.578,Z 328.566,A -85,B 0,C 180,E1 -14340.094,E2 -14340.094} C_VEL
LIN {X 0,Y 340.526,Z 320.88,A -85,B 0,C 180,E1 -14340.616,E2 -14340.616} C_VEL
LIN {X 0,Y 340.338,Z 319.721,A -85,B 0,C 180,E1 -14340.684,E2 -14340.684} C_VEL
LIN {X 0,Y 340.694,Z 315.671,A -85,B 0,C 180,E1 -14344.397,E2 -14344.397} C_VEL
LIN {X 0,Y 341.019,Z 311.703,A -85,B 0,C 180,E1 -14348.189,E2 -14348.189} C_VEL
LIN {X 0,Y 341.221,Z 309.422,A -85,B 0,C 180,E1 -14350.433,E2 -14350.433} C_VEL
LIN {X 0,Y 340.552,Z 308.587,A -85,B 0,C 180,E1 -14351.408,E2 -14351.408} C_VEL
LIN {X 0,Y 337.644,Z 307.519,A -85,B 0,C 180,E1 -14353.001,E2 -14353.001} C_VEL
LIN {X 0,Y 335.154,Z 306.718,A -85,B 0,C 180,E1 -14354.291,E2 -14354.291} C_VEL
LIN {X 0,Y 334.057,Z 305.994,A -85,B 0,C 180,E1 -14355.289,E2 -14355.289} C_VEL
LIN {X 0,Y 333.952,Z 305.711,A -85,B 0,C 180,E1 -14355.626,E2 -14355.626} C_VEL
LIN {X 0,Y 333.707,Z 304.025,A -85,B 0,C 180,E1 -14357.629,E2 -14357.629} C_VEL
LIN {X 0,Y 333.647,Z 303.549,A -85,B 0,C 180,E1 -14359.315,E2 -14359.315} C_VEL
LIN {X 0,Y 333.664,Z 303.551,A -85,B 0,C 180,E1 -14363.168,E2 -14363.168} C_VEL
LIN {X 0,Y 333.673,Z 303.55,A -85,B 0,C 180,E1 -14365.341,E2 -14365.341} C_VEL
LIN {X 0,Y 333.628,Z 303.555,A -85,B 0,C 180,E1 -14368.222,E2 -14368.222} C_VEL
LIN {X 0,Y 333.654,Z 303.549,A -85,B 0,C 180,E1 -14371.022,E2 -14371.022} C_VEL
LIN {X 0,Y 333.697,Z 303.544,A -85,B 0,C 180,E1 -14375.088,E2 -14375.088} C_VEL
LIN {X 0,Y 333.674,Z 303.547,A -85,B 0,C 180,E1 -14379.019,E2 -14379.019} C_VEL
LIN {X 0,Y 333.793,Z 303.531,A -85,B 0,C 180,E1 -14381.589,E2 -14381.589} C_VEL
LIN {X 0,Y 333.807,Z 303.53,A -85,B 0,C 180,E1 -14385.576,E2 -14385.576} C_VEL
LIN {X 0,Y 333.816,Z 303.53,A -85,B 0,C 180,E1 -14389.077,E2 -14389.077} C_VEL
LIN {X 0,Y 333.955,Z 303.512,A -85,B 0,C 180,E1 -14392.746,E2 -14392.746} C_VEL
LIN {X 0,Y 333.8,Z 303.532,A -85,B 0,C 180,E1 -14395.169,E2 -14395.169} C_VEL
LIN {X 0,Y 334.104,Z 303.492,A -85,B 0,C 180,E1 -14397.589,E2 -14397.589} C_VEL
LIN {X 0,Y 334.186,Z 303.484,A -85,B 0,C 180,E1 -14400,E2 -14400} C_VEL
LIN {X 0,Y 334.104,Z 303.493,A -85,B 0,C 180,E1 -14402.411,E2 -14402.411} C_VEL
LIN {X 0,Y 333.99,Z 303.509,A -85,B 0,C 180,E1 -14406.039,E2 -14406.039} C_VEL
LIN {X 0,Y 333.818,Z 303.529,A -85,B 0,C 180,E1 -14409.696,E2 -14409.696} C_VEL
LIN {X 0,Y 333.794,Z 303.533,A -85,B 0,C 180,E1 -14413.391,E2 -14413.391} C_VEL
LIN {X 0,Y 333.744,Z 303.538,A -85,B 0,C 180,E1 -14417.146,E2 -14417.146} C_VEL
LIN {X 0,Y 333.731,Z 303.54,A -85,B 0,C 180,E1 -14419.691,E2 -14419.691} C_VEL
LIN {X 0,Y 333.667,Z 303.547,A -85,B 0,C 180,E1 -14423.59,E2 -14423.59} C_VEL
LIN {X 0,Y 333.733,Z 303.541,A -85,B 0,C 180,E1 -14426.246,E2 -14426.246} C_VEL
LIN {X 0,Y 333.688,Z 303.549,A -85,B 0,C 180,E1 -14428.974,E2 -14428.974} C_VEL
LIN {X 0,Y 333.641,Z 303.558,A -85,B 0,C 180,E1 -14432.587,E2 -14432.587} C_VEL
LIN {X 0,Y 333.674,Z 303.555,A -85,B 0,C 180,E1 -14436.139,E2 -14436.139} C_VEL
LIN {X 0,Y 333.649,Z 303.555,A -85,B 0,C 180,E1 -14438.798,E2 -14438.798} C_VEL
LIN {X 0,Y 334.162,Z 306.989,A -85,B 0,C 180,E1 -14442.599,E2 -14442.599} C_VEL
LIN {X 0,Y 334.624,Z 309.897,A -85,B 0,C 180,E1 -14445.569,E2 -14445.569} C_VEL
LIN {X 0,Y 334.74,Z 312.206,A -85,B 0,C 180,E1 -14447.79,E2 -14447.79} C_VEL
LIN {X 0,Y 334.514,Z 315.777,A -85,B 0,C 180,E1 -14451.019,E2 -14451.019} C_VEL
LIN {X 0,Y 334.121,Z 319.162,A -85,B 0,C 180,E1 -14453.917,E2 -14453.917} C_VEL
LIN {X 0,Y 333.686,Z 323.395,A -85,B 0,C 180,E1 -14457.402,E2 -14457.402} C_VEL
LIN {X 0,Y 333.517,Z 325.169,A -85,B 0,C 180,E1 -14458.681,E2 -14458.681} C_VEL
LIN {X 0,Y 334.501,Z 328.256,A -85,B 0,C 180,E1 -14458.868,E2 -14458.868} C_VEL
LIN {X 0,Y 339.972,Z 343.435,A -85,B 0,C 180,E1 -14459.957,E2 -14459.957} C_VEL
LIN {X 0,Y 343.93,Z 357.615,A -85,B 0,C 180,E1 -14461.066,E2 -14461.066} C_VEL
LIN {X 0,Y 346.775,Z 370.79,A -85,B 0,C 180,E1 -14462.216,E2 -14462.216} C_VEL
LIN {X 0,Y 347.95,Z 378.574,A -85,B 0,C 180,E1 -14462.942,E2 -14462.942} C_VEL
LIN {X 0,Y 345.991,Z 392.366,A -85,B 0,C 180,E1 -14464.105,E2 -14464.105} C_VEL
LIN {X 0,Y 343.764,Z 406.07,A -85,B 0,C 180,E1 -14465.544,E2 -14465.544} C_VEL
LIN {X 0,Y 341.575,Z 418.475,A -85,B 0,C 180,E1 -14467.148,E2 -14467.148} C_VEL
LIN {X 0,Y 339.357,Z 430.664,A -85,B 0,C 180,E1 -14469.074,E2 -14469.074} C_VEL
LIN {X 0,Y 337.547,Z 440.013,A -85,B 0,C 180,E1 -14470.857,E2 -14470.857} C_VEL
LIN {X 0,Y 335.863,Z 449.239,A -85,B 0,C 180,E1 -14472.965,E2 -14472.965} C_VEL
LIN {X 0,Y 334.289,Z 457.922,A -85,B 0,C 180,E1 -14475.387,E2 -14475.387} C_VEL
LIN {X 0,Y 333.304,Z 464.89,A -85,B 0,C 180,E1 -14477.827,E2 -14477.827} C_VEL
LIN {X 0,Y 332.542,Z 470.367,A -85,B 0,C 180,E1 -14480.266,E2 -14480.266} C_VEL
LIN {X 0,Y 332.165,Z 474.507,A -85,B 0,C 180,E1 -14482.706,E2 -14482.706} C_VEL
LIN {X 0,Y 331.941,Z 477.409,A -85,B 0,C 180,E1 -14485.141,E2 -14485.141} C_VEL
LIN {X 0,Y 331.877,Z 479.139,A -85,B 0,C 180,E1 -14487.572,E2 -14487.572} C_VEL
LIN {X 0,Y 331.881,Z 479.732,A -85,B 0,C 180,E1 -14490,E2 -14490} C_VEL
LIN {X 0,Y 331.877,Z 479.132,A -85,B 0,C 180,E1 -14492.427,E2 -14492.427} C_VEL
LIN {X 0,Y 331.95,Z 477.392,A -85,B 0,C 180,E1 -14494.858,E2 -14494.858} C_VEL
LIN {X 0,Y 332.166,Z 474.486,A -85,B 0,C 180,E1 -14497.293,E2 -14497.293} C_VEL
LIN {X 0,Y 332.541,Z 470.344,A -85,B 0,C 180,E1 -14499.733,E2 -14499.733} C_VEL
LIN {X 0,Y 333.301,Z 464.855,A -85,B 0,C 180,E1 -14502.172,E2 -14502.172} C_VEL
LIN {X 0,Y 334.313,Z 457.87,A -85,B 0,C 180,E1 -14504.611,E2 -14504.611} C_VEL
LIN {X 0,Y 335.856,Z 449.179,A -85,B 0,C 180,E1 -14507.034,E2 -14507.034} C_VEL
LIN {X 0,Y 337.553,Z 439.945,A -85,B 0,C 180,E1 -14509.142,E2 -14509.142} C_VEL
LIN {X 0,Y 339.475,Z 430.076,A -85,B 0,C 180,E1 -14511.011,E2 -14511.011} C_VEL
LIN {X 0,Y 341.56,Z 418.376,A -85,B 0,C 180,E1 -14512.853,E2 -14512.853} C_VEL
LIN {X 0,Y 343.703,Z 405.953,A -85,B 0,C 180,E1 -14514.46,E2 -14514.46} C_VEL
LIN {X 0,Y 345.969,Z 392.205,A -85,B 0,C 180,E1 -14515.896,E2 -14515.896} C_VEL
LIN {X 0,Y 347.757,Z 379.645,A -85,B 0,C 180,E1 -14516.963,E2 -14516.963} C_VEL
LIN {X 0,Y 347.713,Z 376.716,A -85,B 0,C 180,E1 -14517.211,E2 -14517.211} C_VEL
LIN {X 0,Y 344.897,Z 361.755,A -85,B 0,C 180,E1 -14518.564,E2 -14518.564} C_VEL
LIN {X 0,Y 340.961,Z 346.716,A -85,B 0,C 180,E1 -14519.776,E2 -14519.776} C_VEL
LIN {X 0,Y 336.079,Z 332.309,A -85,B 0,C 180,E1 -14520.831,E2 -14520.831} C_VEL
LIN {X 0,Y 333.539,Z 325.471,A -85,B 0,C 180,E1 -14521.287,E2 -14521.287} C_VEL
LIN {X 0,Y 333.476,Z 324.959,A -85,B 0,C 180,E1 -14521.339,E2 -14521.339} C_VEL
LIN {X 0,Y 333.959,Z 320.658,A -85,B 0,C 180,E1 -14524.842,E2 -14524.842} C_VEL
LIN {X 0,Y 334.317,Z 317.448,A -85,B 0,C 180,E1 -14527.562,E2 -14527.562} C_VEL
LIN {X 0,Y 334.662,Z 313.673,A -85,B 0,C 180,E1 -14530.886,E2 -14530.886} C_VEL
LIN {X 0,Y 334.675,Z 310.477,A -85,B 0,C 180,E1 -14533.865,E2 -14533.865} C_VEL
LIN {X 0,Y 334.401,Z 308.237,A -85,B 0,C 180,E1 -14536.088,E2 -14536.088} C_VEL
LIN {X 0,Y 333.91,Z 305.216,A -85,B 0,C 180,E1 -14539.272,E2 -14539.272} C_VEL
LIN {X 0,Y 333.645,Z 303.552,A -85,B 0,C 180,E1 -14541.202,E2 -14541.202} C_VEL
LIN {X 0,Y 333.67,Z 303.552,A -85,B 0,C 180,E1 -14543.86,E2 -14543.86} C_VEL
LIN {X 0,Y 333.637,Z 303.558,A -85,B 0,C 180,E1 -14547.413,E2 -14547.413} C_VEL
LIN {X 0,Y 333.683,Z 303.55,A -85,B 0,C 180,E1 -14551.025,E2 -14551.025} C_VEL
LIN {X 0,Y 333.728,Z 303.544,A -85,B 0,C 180,E1 -14553.753,E2 -14553.753} C_VEL
LIN {X 0,Y 333.713,Z 303.541,A -85,B 0,C 180,E1 -14557.914,E2 -14557.914} C_VEL
LIN {X 0,Y 333.787,Z 303.535,A -85,B 0,C 180,E1 -14561.589,E2 -14561.589} C_VEL
LIN {X 0,Y 333.801,Z 303.528,A -85,B 0,C 180,E1 -14565.577,E2 -14565.577} C_VEL
LIN {X 0,Y 333.811,Z 303.529,A -85,B 0,C 180,E1 -14569.077,E2 -14569.077} C_VEL
LIN {X 0,Y 333.95,Z 303.512,A -85,B 0,C 180,E1 -14572.746,E2 -14572.746} C_VEL
LIN {X 0,Y 333.797,Z 303.529,A -85,B 0,C 180,E1 -14575.169,E2 -14575.169} C_VEL
LIN {X 0,Y 334.1,Z 303.488,A -85,B 0,C 180,E1 -14577.589,E2 -14577.589} C_VEL
LIN {X 0,Y 334.2,Z 303.482,A -85,B 0,C 180,E1 -14580,E2 -14580} C_VEL
LIN {X 0,Y 334.1,Z 303.492,A -85,B 0,C 180,E1 -14582.411,E2 -14582.411} C_VEL
LIN {X 0,Y 333.957,Z 303.51,A -85,B 0,C 180,E1 -14586.445,E2 -14586.445} C_VEL
LIN {X 0,Y 333.813,Z 303.529,A -85,B 0,C 180,E1 -14589.697,E2 -14589.697} C_VEL
LIN {X 0,Y 333.79,Z 303.533,A -85,B 0,C 180,E1 -14593.392,E2 -14593.392} C_VEL
LIN {X 0,Y 333.74,Z 303.536,A -85,B 0,C 180,E1 -14597.147,E2 -14597.147} C_VEL
LIN {X 0,Y 333.733,Z 303.54,A -85,B 0,C 180,E1 -14599.691,E2 -14599.691} C_VEL
LIN {X 0,Y 333.686,Z 303.544,A -85,B 0,C 180,E1 -14602.279,E2 -14602.279} C_VEL
LIN {X 0,Y 333.729,Z 303.539,A -85,B 0,C 180,E1 -14606.247,E2 -14606.247} C_VEL
LIN {X 0,Y 333.684,Z 303.543,A -85,B 0,C 180,E1 -14608.975,E2 -14608.975} C_VEL
LIN {X 0,Y 333.638,Z 303.547,A -85,B 0,C 180,E1 -14612.588,E2 -14612.588} C_VEL
LIN {X 0,Y 333.671,Z 303.545,A -85,B 0,C 180,E1 -14616.14,E2 -14616.14} C_VEL
LIN {X 0,Y 333.642,Z 303.552,A -85,B 0,C 180,E1 -14619.193,E2 -14619.193} C_VEL
LIN {X 0,Y 333.642,Z 303.552,A -85,B 0,C 180,E1 -14620.768,E2 -14620.768} C_VEL
LIN {X 0,Y 333.695,Z 304.024,A -85,B 0,C 180,E1 -14622.513,E2 -14622.513} C_VEL
LIN {X 0,Y 334.134,Z 307.045,A -85,B 0,C 180,E1 -14626.046,E2 -14626.046} C_VEL
LIN {X 0,Y 334.196,Z 310.082,A -85,B 0,C 180,E1 -14629.315,E2 -14629.315} C_VEL
LIN {X 0,Y 333.912,Z 313.127,A -85,B 0,C 180,E1 -14632.385,E2 -14632.385} C_VEL
LIN {X 0,Y 333.669,Z 316.184,A -85,B 0,C 180,E1 -14635.342,E2 -14635.342} C_VEL
LIN {X 0,Y 333.325,Z 319.852,A -85,B 0,C 180,E1 -14638.734,E2 -14638.734} C_VEL
LIN {X 0,Y 334.343,Z 323.018,A -85,B 0,C 180,E1 -14638.929,E2 -14638.929} C_VEL
LIN {X 0,Y 339.573,Z 336.496,A -85,B 0,C 180,E1 -14639.926,E2 -14639.926} C_VEL
LIN {X 0,Y 343.626,Z 349.428,A -85,B 0,C 180,E1 -14640.967,E2 -14640.967} C_VEL
LIN {X 0,Y 346.888,Z 362.908,A -85,B 0,C 180,E1 -14642.15,E2 -14642.15} C_VEL
LIN {X 0,Y 348.203,Z 369.66,A -85,B 0,C 180,E1 -14642.79,E2 -14642.79} C_VEL
LIN {X 0,Y 347.882,Z 374.92,A -85,B 0,C 180,E1 -14643.212,E2 -14643.212} C_VEL
LIN {X 0,Y 345.85,Z 388.698,A -85,B 0,C 180,E1 -14644.418,E2 -14644.418} C_VEL
LIN {X 0,Y 343.78,Z 401.925,A -85,B 0,C 180,E1 -14645.867,E2 -14645.867} C_VEL
LIN {X 0,Y 341.804,Z 412.996,A -85,B 0,C 180,E1 -14647.325,E2 -14647.325} C_VEL
LIN {X 0,Y 339.816,Z 424.192,A -85,B 0,C 180,E1 -14649.108,E2 -14649.108} C_VEL
LIN {X 0,Y 337.719,Z 434.981,A -85,B 0,C 180,E1 -14651.183,E2 -14651.183} C_VEL
LIN {X 0,Y 335.984,Z 443.976,A -85,B 0,C 180,E1 -14653.285,E2 -14653.285} C_VEL
LIN {X 0,Y 334.655,Z 451.431,A -85,B 0,C 180,E1 -14655.404,E2 -14655.404} C_VEL
LIN {X 0,Y 333.839,Z 456.792,A -85,B 0,C 180,E1 -14657.23,E2 -14657.23} C_VEL
LIN {X 0,Y 332.898,Z 462.641,A -85,B 0,C 180,E1 -14659.663,E2 -14659.663} C_VEL
LIN {X 0,Y 332.465,Z 466.105,A -85,B 0,C 180,E1 -14661.491,E2 -14661.491} C_VEL
LIN {X 0,Y 332.134,Z 469.704,A -85,B 0,C 180,E1 -14664.003,E2 -14664.003} C_VEL
LIN {X 0,Y 331.996,Z 471.934,A -85,B 0,C 180,E1 -14666.359,E2 -14666.359} C_VEL
LIN {X 0,Y 331.873,Z 473.118,A -85,B 0,C 180,E1 -14668.787,E2 -14668.787} C_VEL
LIN {X 0,Y 331.874,Z 473.133,A -85,B 0,C 180,E1 -14671.214,E2 -14671.214} C_VEL
LIN {X 0,Y 331.996,Z 472.005,A -85,B 0,C 180,E1 -14673.642,E2 -14673.642} C_VEL
LIN {X 0,Y 332.144,Z 469.741,A -85,B 0,C 180,E1 -14676.073,E2 -14676.073} C_VEL
LIN {X 0,Y 332.462,Z 466.283,A -85,B 0,C 180,E1 -14678.51,E2 -14678.51} C_VEL
LIN {X 0,Y 333.033,Z 461.551,A -85,B 0,C 180,E1 -14680.949,E2 -14680.949} C_VEL
LIN {X 0,Y 334.082,Z 455.419,A -85,B 0,C 180,E1 -14683.38,E2 -14683.38} C_VEL
LIN {X 0,Y 335.323,Z 447.702,A -85,B 0,C 180,E1 -14685.811,E2 -14685.811} C_VEL
LIN {X 0,Y 336.861,Z 439.475,A -85,B 0,C 180,E1 -14687.923,E2 -14687.923} C_VEL
LIN {X 0,Y 338.761,Z 429.565,A -85,B 0,C 180,E1 -14690.018,E2 -14690.018} C_VEL
LIN {X 0,Y 340.689,Z 419.228,A -85,B 0,C 180,E1 -14691.829,E2 -14691.829} C_VEL
LIN {X 0,Y 342.814,Z 407.314,A -85,B 0,C 180,E1 -14693.564,E2 -14693.564} C_VEL
LIN {X 0,Y 344.847,Z 395.189,A -85,B 0,C 180,E1 -14695.017,E2 -14695.017} C_VEL
LIN {X 0,Y 346.948,Z 382.012,A -85,B 0,C 180,E1 -14696.303,E2 -14696.303} C_VEL
LIN {X 0,Y 348.362,Z 370.627,A -85,B 0,C 180,E1 -14697.225,E2 -14697.225} C_VEL
LIN {X 0,Y 345.586,Z 357.109,A -85,B 0,C 180,E1 -14698.485,E2 -14698.485} C_VEL
LIN {X 0,Y 342.11,Z 344.212,A -85,B 0,C 180,E1 -14699.573,E2 -14699.573} C_VEL
LIN {X 0,Y 337.116,Z 329.8,A -85,B 0,C 180,E1 -14700.688,E2 -14700.688} C_VEL
LIN {X 0,Y 333.424,Z 320.466,A -85,B 0,C 180,E1 -14701.353,E2 -14701.353} C_VEL
LIN {X 0,Y 333.338,Z 319.773,A -85,B 0,C 180,E1 -14701.425,E2 -14701.425} C_VEL
LIN {X 0,Y 333.682,Z 316.217,A -85,B 0,C 180,E1 -14704.773,E2 -14704.773} C_VEL
LIN {X 0,Y 333.912,Z 313.277,A -85,B 0,C 180,E1 -14707.617,E2 -14707.617} C_VEL
LIN {X 0,Y 334.209,Z 310.14,A -85,B 0,C 180,E1 -14710.796,E2 -14710.796} C_VEL
LIN {X 0,Y 334.162,Z 307.184,A -85,B 0,C 180,E1 -14713.951,E2 -14713.951} C_VEL
LIN {X 0,Y 333.952,Z 305.711,A -85,B 0,C 180,E1 -14715.626,E2 -14715.626} C_VEL
LIN {X 0,Y 333.216,Z 305.014,A -85,B 0,C 180,E1 -14716.624,E2 -14716.624} C_VEL
LIN {X 0,Y 330.239,Z 304.485,A -85,B 0,C 180,E1 -14718.253,E2 -14718.253} C_VEL
LIN {X 0,Y 327.749,Z 304.411,A -85,B 0,C 180,E1 -14719.578,E2 -14719.578} C_VEL
LIN {X 0,Y 326.692,Z 304.426,A -85,B 0,C 180,E1 -14720.605,E2 -14720.605} C_VEL
LIN {X 0,Y 326.61,Z 304.428,A -85,B 0,C 180,E1 -14720.953,E2 -14720.953} C_VEL
LIN {X 0,Y 326.612,Z 304.429,A -85,B 0,C 180,E1 -14724.48,E2 -14724.48} C_VEL
LIN {X 0,Y 326.607,Z 304.429,A -85,B 0,C 180,E1 -14727.455,E2 -14727.455} C_VEL
LIN {X 0,Y 326.616,Z 304.427,A -85,B 0,C 180,E1 -14730.336,E2 -14730.336} C_VEL
LIN {X 0,Y 326.641,Z 304.422,A -85,B 0,C 180,E1 -14734.644,E2 -14734.644} C_VEL
LIN {X 0,Y 326.619,Z 304.424,A -85,B 0,C 180,E1 -14738.543,E2 -14738.543} C_VEL
LIN {X 0,Y 326.743,Z 304.407,A -85,B 0,C 180,E1 -14741.177,E2 -14741.177} C_VEL
LIN {X 0,Y 326.762,Z 304.408,A -85,B 0,C 180,E1 -14745.433,E2 -14745.433} C_VEL
LIN {X 0,Y 326.756,Z 304.408,A -85,B 0,C 180,E1 -14748.838,E2 -14748.838} C_VEL
LIN {X 0,Y 326.912,Z 304.39,A -85,B 0,C 180,E1 -14752.589,E2 -14752.589} C_VEL
LIN {X 0,Y 326.767,Z 304.408,A -85,B 0,C 180,E1 -14755.065,E2 -14755.065} C_VEL
LIN {X 0,Y 327.045,Z 304.372,A -85,B 0,C 180,E1 -14757.537,E2 -14757.537} C_VEL
LIN {X 0,Y 327.139,Z 304.362,A -85,B 0,C 180,E1 -14760,E2 -14760} C_VEL
LIN {X 0,Y 327.045,Z 304.372,A -85,B 0,C 180,E1 -14762.463,E2 -14762.463} C_VEL
LIN {X 0,Y 326.944,Z 304.387,A -85,B 0,C 180,E1 -14766.17,E2 -14766.17} C_VEL
LIN {X 0,Y 326.781,Z 304.405,A -85,B 0,C 180,E1 -14769.907,E2 -14769.907} C_VEL
LIN {X 0,Y 326.757,Z 304.411,A -85,B 0,C 180,E1 -14773.685,E2 -14773.685} C_VEL
LIN {X 0,Y 326.697,Z 304.415,A -85,B 0,C 180,E1 -14777.528,E2 -14777.528} C_VEL
LIN {X 0,Y 326.657,Z 304.422,A -85,B 0,C 180,E1 -14780.135,E2 -14780.135} C_VEL
LIN {X 0,Y 326.647,Z 304.422,A -85,B 0,C 180,E1 -14784.129,E2 -14784.129} C_VEL
LIN {X 0,Y 326.681,Z 304.419,A -85,B 0,C 180,E1 -14786.858,E2 -14786.858} C_VEL
LIN {X 0,Y 326.632,Z 304.43,A -85,B 0,C 180,E1 -14790.61,E2 -14790.61} C_VEL
LIN {X 0,Y 326.605,Z 304.436,A -85,B 0,C 180,E1 -14794.019,E2 -14794.019} C_VEL
LIN {X 0,Y 326.625,Z 304.433,A -85,B 0,C 180,E1 -14797.238,E2 -14797.238} C_VEL
LIN {X 0,Y 326.646,Z 304.632,A -85,B 0,C 180,E1 -14798.605,E2 -14798.605} C_VEL
LIN {X 0,Y 327.057,Z 307.426,A -85,B 0,C 180,E1 -14801.77,E2 -14801.77} C_VEL
LIN {X 0,Y 327.571,Z 310.546,A -85,B 0,C 180,E1 -14805.073,E2 -14805.073} C_VEL
LIN {X 0,Y 327.668,Z 313.892,A -85,B 0,C 180,E1 -14808.325,E2 -14808.325} C_VEL
LIN {X 0,Y 327.4,Z 317.345,A -85,B 0,C 180,E1 -14811.5,E2 -14811.5} C_VEL
LIN {X 0,Y 326.952,Z 321.131,A -85,B 0,C 180,E1 -14814.768,E2 -14814.768} C_VEL
LIN {X 0,Y 326.534,Z 324.893,A -85,B 0,C 180,E1 -14817.918,E2 -14817.918} C_VEL
LIN {X 0,Y 327.584,Z 328.233,A -85,B 0,C 180,E1 -14818.136,E2 -14818.136} C_VEL
LIN {X 0,Y 333.063,Z 343.2,A -85,B 0,C 180,E1 -14819.259,E2 -14819.259} C_VEL
LIN {X 0,Y 337.165,Z 357.531,A -85,B 0,C 180,E1 -14820.427,E2 -14820.427} C_VEL
LIN {X 0,Y 340.009,Z 370.723,A -85,B 0,C 180,E1 -14821.614,E2 -14821.614} C_VEL
LIN {X 0,Y 341.454,Z 379.672,A -85,B 0,C 180,E1 -14822.487,E2 -14822.487} C_VEL
LIN {X 0,Y 339.371,Z 393.809,A -85,B 0,C 180,E1 -14823.727,E2 -14823.727} C_VEL
LIN {X 0,Y 337.063,Z 407.214,A -85,B 0,C 180,E1 -14825.189,E2 -14825.189} C_VEL
LIN {X 0,Y 334.798,Z 419.422,A -85,B 0,C 180,E1 -14826.821,E2 -14826.821} C_VEL
LIN {X 0,Y 332.609,Z 430.929,A -85,B 0,C 180,E1 -14828.695,E2 -14828.695} C_VEL
LIN {X 0,Y 330.507,Z 441.38,A -85,B 0,C 180,E1 -14830.756,E2 -14830.756} C_VEL
LIN {X 0,Y 328.798,Z 450.386,A -85,B 0,C 180,E1 -14832.908,E2 -14832.908} C_VEL
LIN {X 0,Y 327.351,Z 457.854,A -85,B 0,C 180,E1 -14835.07,E2 -14835.07} C_VEL
LIN {X 0,Y 326.304,Z 464.821,A -85,B 0,C 180,E1 -14837.562,E2 -14837.562} C_VEL
LIN {X 0,Y 325.49,Z 470.298,A -85,B 0,C 180,E1 -14840.053,E2 -14840.053} C_VEL
LIN {X 0,Y 325.079,Z 474.439,A -85,B 0,C 180,E1 -14842.546,E2 -14842.546} C_VEL
LIN {X 0,Y 324.856,Z 477.341,A -85,B 0,C 180,E1 -14845.035,E2 -14845.035} C_VEL
LIN {X 0,Y 324.798,Z 479.071,A -85,B 0,C 180,E1 -14847.519,E2 -14847.519} C_VEL
LIN {X 0,Y 324.79,Z 479.663,A -85,B 0,C 180,E1 -14850,E2 -14850} C_VEL
LIN {X 0,Y 324.798,Z 479.063,A -85,B 0,C 180,E1 -14852.48,E2 -14852.48} C_VEL
LIN {X 0,Y 324.864,Z 477.323,A -85,B 0,C 180,E1 -14854.964,E2 -14854.964} C_VEL
LIN {X 0,Y 325.079,Z 474.416,A -85,B 0,C 180,E1 -14857.453,E2 -14857.453} C_VEL
LIN {X 0,Y 325.489,Z 470.273,A -85,B 0,C 180,E1 -14859.946,E2 -14859.946} C_VEL
LIN {X 0,Y 326.301,Z 464.785,A -85,B 0,C 180,E1 -14862.437,E2 -14862.437} C_VEL
LIN {X 0,Y 327.402,Z 457.595,A -85,B 0,C 180,E1 -14864.991,E2 -14864.991} C_VEL
LIN {X 0,Y 329.019,Z 449.108,A -85,B 0,C 180,E1 -14867.4,E2 -14867.4} C_VEL
LIN {X 0,Y 330.794,Z 439.873,A -85,B 0,C 180,E1 -14869.549,E2 -14869.549} C_VEL
LIN {X 0,Y 332.661,Z 430.689,A -85,B 0,C 180,E1 -14871.332,E2 -14871.332} C_VEL
LIN {X 0,Y 334.786,Z 419.327,A -85,B 0,C 180,E1 -14873.178,E2 -14873.178} C_VEL
LIN {X 0,Y 336.997,Z 407.101,A -85,B 0,C 180,E1 -14874.815,E2 -14874.815} C_VEL
LIN {X 0,Y 339.345,Z 393.656,A -85,B 0,C 180,E1 -14876.274,E2 -14876.274} C_VEL
LIN {X 0,Y 341.382,Z 379.57,A -85,B 0,C 180,E1 -14877.509,E2 -14877.509} C_VEL
LIN {X 0,Y 338.888,Z 365.104,A -85,B 0,C 180,E1 -14878.889,E2 -14878.889} C_VEL
LIN {X 0,Y 335.023,Z 349.713,A -85,B 0,C 180,E1 -14880.209,E2 -14880.209} C_VEL
LIN {X 0,Y 330.798,Z 336.837,A -85,B 0,C 180,E1 -14881.214,E2 -14881.214} C_VEL
LIN {X 0,Y 326.608,Z 325.521,A -85,B 0,C 180,E1 -14882.025,E2 -14882.025} C_VEL
LIN {X 0,Y 326.523,Z 324.883,A -85,B 0,C 180,E1 -14882.084,E2 -14882.084} C_VEL
LIN {X 0,Y 326.977,Z 320.852,A -85,B 0,C 180,E1 -14885.473,E2 -14885.473} C_VEL
LIN {X 0,Y 327.396,Z 317.374,A -85,B 0,C 180,E1 -14888.499,E2 -14888.499} C_VEL
LIN {X 0,Y 327.668,Z 313.898,A -85,B 0,C 180,E1 -14891.674,E2 -14891.674} C_VEL
LIN {X 0,Y 327.569,Z 310.556,A -85,B 0,C 180,E1 -14894.926,E2 -14894.926} C_VEL
LIN {X 0,Y 326.974,Z 306.903,A -85,B 0,C 180,E1 -14898.788,E2 -14898.788} C_VEL
LIN {X 0,Y 326.642,Z 304.594,A -85,B 0,C 180,E1 -14901.394,E2 -14901.394} C_VEL
LIN {X 0,Y 326.613,Z 304.432,A -85,B 0,C 180,E1 -14904.851,E2 -14904.851} C_VEL
LIN {X 0,Y 326.601,Z 304.435,A -85,B 0,C 180,E1 -14907.455,E2 -14907.455} C_VEL
LIN {X 0,Y 326.641,Z 304.428,A -85,B 0,C 180,E1 -14910.339,E2 -14910.339} C_VEL
LIN {X 0,Y 326.683,Z 304.418,A -85,B 0,C 180,E1 -14914.516,E2 -14914.516} C_VEL
LIN {X 0,Y 326.642,Z 304.422,A -85,B 0,C 180,E1 -14918.545,E2 -14918.545} C_VEL
LIN {X 0,Y 326.738,Z 304.41,A -85,B 0,C 180,E1 -14921.177,E2 -14921.177} C_VEL
LIN {X 0,Y 326.756,Z 304.405,A -85,B 0,C 180,E1 -14925.433,E2 -14925.433} C_VEL
LIN {X 0,Y 326.751,Z 304.407,A -85,B 0,C 180,E1 -14928.838,E2 -14928.838} C_VEL
LIN {X 0,Y 326.906,Z 304.391,A -85,B 0,C 180,E1 -14932.589,E2 -14932.589} C_VEL
LIN {X 0,Y 326.763,Z 304.405,A -85,B 0,C 180,E1 -14935.065,E2 -14935.065} C_VEL
LIN {X 0,Y 327.041,Z 304.367,A -85,B 0,C 180,E1 -14937.537,E2 -14937.537} C_VEL
LIN {X 0,Y 327.152,Z 304.36,A -85,B 0,C 180,E1 -14940,E2 -14940} C_VEL
LIN {X 0,Y 327.041,Z 304.372,A -85,B 0,C 180,E1 -14942.463,E2 -14942.463} C_VEL
LIN {X 0,Y 326.919,Z 304.387,A -85,B 0,C 180,E1 -14946.432,E2 -14946.432} C_VEL
LIN {X 0,Y 326.776,Z 304.406,A -85,B 0,C 180,E1 -14949.908,E2 -14949.908} C_VEL
LIN {X 0,Y 326.752,Z 304.41,A -85,B 0,C 180,E1 -14953.686,E2 -14953.686} C_VEL
LIN {X 0,Y 326.692,Z 304.413,A -85,B 0,C 180,E1 -14957.528,E2 -14957.528} C_VEL
LIN {X 0,Y 326.659,Z 304.419,A -85,B 0,C 180,E1 -14960.135,E2 -14960.135} C_VEL
LIN {X 0,Y 326.646,Z 304.422,A -85,B 0,C 180,E1 -14964.129,E2 -14964.129} C_VEL
LIN {X 0,Y 326.677,Z 304.416,A -85,B 0,C 180,E1 -14966.858,E2 -14966.858} C_VEL
LIN {X 0,Y 326.628,Z 304.422,A -85,B 0,C 180,E1 -14970.61,E2 -14970.61} C_VEL
LIN {X 0,Y 326.601,Z 304.424,A -85,B 0,C 180,E1 -14974.02,E2 -14974.02} C_VEL
LIN {X 0,Y 326.623,Z 304.424,A -85,B 0,C 180,E1 -14977.239,E2 -14977.239} C_VEL
LIN {X 0,Y 326.573,Z 304.432,A -85,B 0,C 180,E1 -14981.132,E2 -14981.132} C_VEL
LIN {X 0,Y 326.597,Z 304.665,A -85,B 0,C 180,E1 -14981.843,E2 -14981.843} C_VEL
LIN {X 0,Y 327.016,Z 307.412,A -85,B 0,C 180,E1 -14985.171,E2 -14985.171} C_VEL
LIN {X 0,Y 327.178,Z 310.155,A -85,B 0,C 180,E1 -14988.25,E2 -14988.25} C_VEL
LIN {X 0,Y 326.981,Z 313.204,A -85,B 0,C 180,E1 -14991.443,E2 -14991.443} C_VEL
LIN {X 0,Y 326.677,Z 316.599,A -85,B 0,C 180,E1 -14994.837,E2 -14994.837} C_VEL
LIN {X 0,Y 326.34,Z 319.865,A -85,B 0,C 180,E1 -14997.964,E2 -14997.964} C_VEL
LIN {X 0,Y 327.37,Z 323.073,A -85,B 0,C 180,E1 -14998.189,E2 -14998.189} C_VEL
LIN {X 0,Y 332.949,Z 337.29,A -85,B 0,C 180,E1 -14999.297,E2 -14999.297} C_VEL
LIN {X 0,Y 337.26,Z 351.166,A -85,B 0,C 180,E1 -15000.459,E2 -15000.459} C_VEL
LIN {X 0,Y 339.97,Z 362.204,A -85,B 0,C 180,E1 -15001.473,E2 -15001.473} C_VEL
LIN {X 0,Y 341.771,Z 371.602,A -85,B 0,C 180,E1 -15002.391,E2 -15002.391} C_VEL
LIN {X 0,Y 340.441,Z 382.622,A -85,B 0,C 180,E1 -15003.321,E2 -15003.321} C_VEL
LIN {X 0,Y 338.34,Z 395.708,A -85,B 0,C 180,E1 -15004.633,E2 -15004.633} C_VEL
LIN {X 0,Y 336.224,Z 407.757,A -85,B 0,C 180,E1 -15006.11,E2 -15006.11} C_VEL
LIN {X 0,Y 334.17,Z 418.888,A -85,B 0,C 180,E1 -15007.756,E2 -15007.756} C_VEL
LIN {X 0,Y 332.137,Z 429.105,A -85,B 0,C 180,E1 -15009.566,E2 -15009.566} C_VEL
LIN {X 0,Y 330.133,Z 439.102,A -85,B 0,C 180,E1 -15011.7,E2 -15011.7} C_VEL
LIN {X 0,Y 328.506,Z 447.395,A -85,B 0,C 180,E1 -15013.853,E2 -15013.853} C_VEL
LIN {X 0,Y 327.171,Z 455.184,A -85,B 0,C 180,E1 -15016.333,E2 -15016.333} C_VEL
LIN {X 0,Y 326.036,Z 461.386,A -85,B 0,C 180,E1 -15018.814,E2 -15018.814} C_VEL
LIN {X 0,Y 325.426,Z 466.175,A -85,B 0,C 180,E1 -15021.306,E2 -15021.306} C_VEL
LIN {X 0,Y 325.024,Z 470.012,A -85,B 0,C 180,E1 -15024.077,E2 -15024.077} C_VEL
LIN {X 0,Y 324.903,Z 472.003,A -85,B 0,C 180,E1 -15026.28,E2 -15026.28} C_VEL
LIN {X 0,Y 324.785,Z 473.187,A -85,B 0,C 180,E1 -15028.761,E2 -15028.761} C_VEL
LIN {X 0,Y 324.785,Z 473.201,A -85,B 0,C 180,E1 -15031.24,E2 -15031.24} C_VEL
LIN {X 0,Y 324.902,Z 472.074,A -85,B 0,C 180,E1 -15033.721,E2 -15033.721} C_VEL
LIN {X 0,Y 325.055,Z 469.809,A -85,B 0,C 180,E1 -15036.206,E2 -15036.206} C_VEL
LIN {X 0,Y 325.422,Z 466.351,A -85,B 0,C 180,E1 -15038.695,E2 -15038.695} C_VEL
LIN {X 0,Y 326.011,Z 461.619,A -85,B 0,C 180,E1 -15041.188,E2 -15041.188} C_VEL
LIN {X 0,Y 327.128,Z 455.487,A -85,B 0,C 180,E1 -15043.67,E2 -15043.67} C_VEL
LIN {X 0,Y 328.444,Z 447.769,A -85,B 0,C 180,E1 -15046.151,E2 -15046.151} C_VEL
LIN {X 0,Y 330.063,Z 439.542,A -85,B 0,C 180,E1 -15048.305,E2 -15048.305} C_VEL
LIN {X 0,Y 332.077,Z 429.632,A -85,B 0,C 180,E1 -15050.439,E2 -15050.439} C_VEL
LIN {X 0,Y 334.04,Z 419.474,A -85,B 0,C 180,E1 -15052.254,E2 -15052.254} C_VEL
LIN {X 0,Y 336.31,Z 407.379,A -85,B 0,C 180,E1 -15054.048,E2 -15054.048} C_VEL
LIN {X 0,Y 338.409,Z 395.253,A -85,B 0,C 180,E1 -15055.527,E2 -15055.527} C_VEL
LIN {X 0,Y 340.578,Z 382.076,A -85,B 0,C 180,E1 -15056.834,E2 -15056.834} C_VEL
LIN {X 0,Y 341.897,Z 372.001,A -85,B 0,C 180,E1 -15057.674,E2 -15057.674} C_VEL
LIN {X 0,Y 339.071,Z 358.101,A -85,B 0,C 180,E1 -15059.023,E2 -15059.023} C_VEL
LIN {X 0,Y 335.042,Z 343.581,A -85,B 0,C 180,E1 -15060.3,E2 -15060.3} C_VEL
LIN {X 0,Y 329.896,Z 329.149,A -85,B 0,C 180,E1 -15061.463,E2 -15061.463} C_VEL
LIN {X 0,Y 326.445,Z 320.508,A -85,B 0,C 180,E1 -15062.103,E2 -15062.103} C_VEL
LIN {X 0,Y 326.359,Z 319.886,A -85,B 0,C 180,E1 -15062.144,E2 -15062.144} C_VEL
LIN {X 0,Y 326.705,Z 316.388,A -85,B 0,C 180,E1 -15065.508,E2 -15065.508} C_VEL
LIN {X 0,Y 327.058,Z 312.613,A -85,B 0,C 180,E1 -15069.323,E2 -15069.323} C_VEL
LIN {X 0,Y 327.19,Z 310.295,A -85,B 0,C 180,E1 -15071.749,E2 -15071.749} C_VEL
LIN {X 0,Y 327.036,Z 307.545,A -85,B 0,C 180,E1 -15074.832,E2 -15074.832} C_VEL
LIN {X 0,Y 326.645,Z 304.773,A -85,B 0,C 180,E1 -15078.165,E2 -15078.165} C_VEL
LIN {X 0,Y 326.591,Z 304.427,A -85,B 0,C 180,E1 -15079.791,E2 -15079.791} C_VEL
LIN {X 0,Y 326.61,Z 304.428,A -85,B 0,C 180,E1 -15080.953,E2 -15080.953} C_VEL
LIN {X 0,Y 325.943,Z 304.513,A -85,B 0,C 180,E1 -15081.983,E2 -15081.983} C_VEL
LIN {X 0,Y 323.054,Z 304.874,A -85,B 0,C 180,E1 -15083.659,E2 -15083.659} C_VEL
LIN {X 0,Y 320.626,Z 305.176,A -85,B 0,C 180,E1 -15085.017,E2 -15085.017} C_VEL
LIN {X 0,Y 319.621,Z 305.299,A -85,B 0,C 180,E1 -15086.069,E2 -15086.069} C_VEL
LIN {X 0,Y 319.559,Z 305.307,A -85,B 0,C 180,E1 -15086.425,E2 -15086.425} C_VEL
LIN {X 0,Y 319.559,Z 305.305,A -85,B 0,C 180,E1 -15089.613,E2 -15089.613} C_VEL
LIN {X 0,Y 319.545,Z 305.308,A -85,B 0,C 180,E1 -15092.492,E2 -15092.492} C_VEL
LIN {X 0,Y 319.573,Z 305.302,A -85,B 0,C 180,E1 -15095.301,E2 -15095.301} C_VEL
LIN {X 0,Y 319.602,Z 305.299,A -85,B 0,C 180,E1 -15099.4,E2 -15099.4} C_VEL
LIN {X 0,Y 319.657,Z 305.293,A -85,B 0,C 180,E1 -15102.073,E2 -15102.073} C_VEL
LIN {X 0,Y 319.73,Z 305.284,A -85,B 0,C 180,E1 -15106.008,E2 -15106.008} C_VEL
LIN {X 0,Y 319.733,Z 305.283,A -85,B 0,C 180,E1 -15109.872,E2 -15109.872} C_VEL
LIN {X 0,Y 319.9,Z 305.262,A -85,B 0,C 180,E1 -15113.693,E2 -15113.693} C_VEL
LIN {X 0,Y 319.989,Z 305.251,A -85,B 0,C 180,E1 -15117.482,E2 -15117.482} C_VEL
LIN {X 0,Y 320.093,Z 305.239,A -85,B 0,C 180,E1 -15120,E2 -15120} C_VEL
LIN {X 0,Y 319.989,Z 305.251,A -85,B 0,C 180,E1 -15122.517,E2 -15122.517} C_VEL
LIN {X 0,Y 319.9,Z 305.263,A -85,B 0,C 180,E1 -15126.306,E2 -15126.306} C_VEL
LIN {X 0,Y 319.733,Z 305.283,A -85,B 0,C 180,E1 -15130.128,E2 -15130.128} C_VEL
LIN {X 0,Y 319.73,Z 305.284,A -85,B 0,C 180,E1 -15133.992,E2 -15133.992} C_VEL
LIN {X 0,Y 319.656,Z 305.292,A -85,B 0,C 180,E1 -15137.927,E2 -15137.927} C_VEL
LIN {X 0,Y 319.6,Z 305.299,A -85,B 0,C 180,E1 -15140.6,E2 -15140.6} C_VEL
LIN {X 0,Y 319.601,Z 305.301,A -85,B 0,C 180,E1 -15144.696,E2 -15144.696} C_VEL
LIN {X 0,Y 319.609,Z 305.302,A -85,B 0,C 180,E1 -15148.41,E2 -15148.41} C_VEL
LIN {X 0,Y 319.529,Z 305.315,A -85,B 0,C 180,E1 -15151.862,E2 -15151.862} C_VEL
LIN {X 0,Y 319.578,Z 305.312,A -85,B 0,C 180,E1 -15155.543,E2 -15155.543} C_VEL
LIN {X 0,Y 319.582,Z 305.424,A -85,B 0,C 180,E1 -15158.007,E2 -15158.007} C_VEL
LIN {X 0,Y 320.057,Z 308.599,A -85,B 0,C 180,E1 -15161.704,E2 -15161.704} C_VEL
LIN {X 0,Y 320.578,Z 312.082,A -85,B 0,C 180,E1 -15165.45,E2 -15165.45} C_VEL
LIN {X 0,Y 320.667,Z 314.819,A -85,B 0,C 180,E1 -15168.174,E2 -15168.174} C_VEL
LIN {X 0,Y 320.499,Z 317.303,A -85,B 0,C 180,E1 -15170.512,E2 -15170.512} C_VEL
LIN {X 0,Y 320.069,Z 320.766,A -85,B 0,C 180,E1 -15173.64,E2 -15173.64} C_VEL
LIN {X 0,Y 319.613,Z 324.839,A -85,B 0,C 180,E1 -15177.146,E2 -15177.146} C_VEL
LIN {X 0,Y 320.706,Z 328.25,A -85,B 0,C 180,E1 -15177.371,E2 -15177.371} C_VEL
LIN {X 0,Y 326.078,Z 342.723,A -85,B 0,C 180,E1 -15178.506,E2 -15178.506} C_VEL
LIN {X 0,Y 330.155,Z 356.445,A -85,B 0,C 180,E1 -15179.67,E2 -15179.67} C_VEL
LIN {X 0,Y 333.029,Z 369.26,A -85,B 0,C 180,E1 -15180.857,E2 -15180.857} C_VEL
LIN {X 0,Y 334.926,Z 380.732,A -85,B 0,C 180,E1 -15182.012,E2 -15182.012} C_VEL
LIN {X 0,Y 332.998,Z 393.743,A -85,B 0,C 180,E1 -15183.184,E2 -15183.184} C_VEL
LIN {X 0,Y 330.595,Z 407.148,A -85,B 0,C 180,E1 -15184.67,E2 -15184.67} C_VEL
LIN {X 0,Y 328.224,Z 419.355,A -85,B 0,C 180,E1 -15186.329,E2 -15186.329} C_VEL
LIN {X 0,Y 326.032,Z 430.234,A -85,B 0,C 180,E1 -15188.118,E2 -15188.118} C_VEL
LIN {X 0,Y 324.072,Z 439.878,A -85,B 0,C 180,E1 -15190.028,E2 -15190.028} C_VEL
LIN {X 0,Y 322.189,Z 449.103,A -85,B 0,C 180,E1 -15192.218,E2 -15192.218} C_VEL
LIN {X 0,Y 320.445,Z 457.785,A -85,B 0,C 180,E1 -15194.741,E2 -15194.741} C_VEL
LIN {X 0,Y 319.319,Z 464.753,A -85,B 0,C 180,E1 -15197.285,E2 -15197.285} C_VEL
LIN {X 0,Y 318.457,Z 470.229,A -85,B 0,C 180,E1 -15199.831,E2 -15199.831} C_VEL
LIN {X 0,Y 318.003,Z 474.37,A -85,B 0,C 180,E1 -15202.38,E2 -15202.38} C_VEL
LIN {X 0,Y 317.774,Z 477.272,A -85,B 0,C 180,E1 -15204.924,E2 -15204.924} C_VEL
LIN {X 0,Y 317.721,Z 479.002,A -85,B 0,C 180,E1 -15207.464,E2 -15207.464} C_VEL
LIN {X 0,Y 317.701,Z 479.594,A -85,B 0,C 180,E1 -15210,E2 -15210} C_VEL
LIN {X 0,Y 317.721,Z 478.994,A -85,B 0,C 180,E1 -15212.535,E2 -15212.535} C_VEL
LIN {X 0,Y 317.782,Z 477.253,A -85,B 0,C 180,E1 -15215.075,E2 -15215.075} C_VEL
LIN {X 0,Y 318.004,Z 474.346,A -85,B 0,C 180,E1 -15217.619,E2 -15217.619} C_VEL
LIN {X 0,Y 318.456,Z 470.203,A -85,B 0,C 180,E1 -15220.168,E2 -15220.168} C_VEL
LIN {X 0,Y 319.316,Z 464.714,A -85,B 0,C 180,E1 -15222.714,E2 -15222.714} C_VEL
LIN {X 0,Y 320.445,Z 457.728,A -85,B 0,C 180,E1 -15225.258,E2 -15225.258} C_VEL
LIN {X 0,Y 322.18,Z 449.036,A -85,B 0,C 180,E1 -15227.781,E2 -15227.781} C_VEL
LIN {X 0,Y 324.08,Z 439.801,A -85,B 0,C 180,E1 -15229.971,E2 -15229.971} C_VEL
LIN {X 0,Y 326.118,Z 429.769,A -85,B 0,C 180,E1 -15231.945,E2 -15231.945} C_VEL
LIN {X 0,Y 328.442,Z 418.231,A -85,B 0,C 180,E1 -15233.821,E2 -15233.821} C_VEL
LIN {X 0,Y 330.766,Z 405.807,A -85,B 0,C 180,E1 -15235.483,E2 -15235.483} C_VEL
LIN {X 0,Y 333.216,Z 392.057,A -85,B 0,C 180,E1 -15236.965,E2 -15236.965} C_VEL
LIN {X 0,Y 334.876,Z 380.73,A -85,B 0,C 180,E1 -15237.971,E2 -15237.971} C_VEL
LIN {X 0,Y 332.563,Z 367.002,A -85,B 0,C 180,E1 -15239.34,E2 -15239.34} C_VEL
LIN {X 0,Y 329.043,Z 352.623,A -85,B 0,C 180,E1 -15240.643,E2 -15240.643} C_VEL
LIN {X 0,Y 324.908,Z 339.505,A -85,B 0,C 180,E1 -15241.736,E2 -15241.736} C_VEL
LIN {X 0,Y 319.724,Z 325.648,A -85,B 0,C 180,E1 -15242.793,E2 -15242.793} C_VEL
LIN {X 0,Y 319.594,Z 324.822,A -85,B 0,C 180,E1 -15242.854,E2 -15242.854} C_VEL
LIN {X 0,Y 320.055,Z 320.778,A -85,B 0,C 180,E1 -15246.361,E2 -15246.361} C_VEL
LIN {X 0,Y 320.521,Z 316.887,A -85,B 0,C 180,E1 -15249.876,E2 -15249.876} C_VEL
LIN {X 0,Y 320.664,Z 313.826,A -85,B 0,C 180,E1 -15252.797,E2 -15252.797} C_VEL
LIN {X 0,Y 320.47,Z 311.236,A -85,B 0,C 180,E1 -15255.431,E2 -15255.431} C_VEL
LIN {X 0,Y 320.002,Z 308.137,A -85,B 0,C 180,E1 -15258.786,E2 -15258.786} C_VEL
LIN {X 0,Y 319.578,Z 305.383,A -85,B 0,C 180,E1 -15261.993,E2 -15261.993} C_VEL
LIN {X 0,Y 319.554,Z 305.312,A -85,B 0,C 180,E1 -15265.123,E2 -15265.123} C_VEL
LIN {X 0,Y 319.56,Z 305.312,A -85,B 0,C 180,E1 -15269.059,E2 -15269.059} C_VEL
LIN {X 0,Y 319.599,Z 305.303,A -85,B 0,C 180,E1 -15272.497,E2 -15272.497} C_VEL
LIN {X 0,Y 319.598,Z 305.302,A -85,B 0,C 180,E1 -15275.304,E2 -15275.304} C_VEL
LIN {X 0,Y 319.591,Z 305.301,A -85,B 0,C 180,E1 -15278.048,E2 -15278.048} C_VEL
LIN {X 0,Y 319.683,Z 305.288,A -85,B 0,C 180,E1 -15280.962,E2 -15280.962} C_VEL
LIN {X 0,Y 319.724,Z 305.281,A -85,B 0,C 180,E1 -15285.276,E2 -15285.276} C_VEL
LIN {X 0,Y 319.708,Z 305.284,A -85,B 0,C 180,E1 -15288.589,E2 -15288.589} C_VEL
LIN {X 0,Y 319.846,Z 305.271,A -85,B 0,C 180,E1 -15292.424,E2 -15292.424} C_VEL
LIN {X 0,Y 319.73,Z 305.28,A -85,B 0,C 180,E1 -15294.956,E2 -15294.956} C_VEL
LIN {X 0,Y 319.984,Z 305.246,A -85,B 0,C 180,E1 -15297.482,E2 -15297.482} C_VEL
LIN {X 0,Y 320.105,Z 305.238,A -85,B 0,C 180,E1 -15300,E2 -15300} C_VEL
LIN {X 0,Y 319.984,Z 305.251,A -85,B 0,C 180,E1 -15302.518,E2 -15302.518} C_VEL
LIN {X 0,Y 319.885,Z 305.265,A -85,B 0,C 180,E1 -15306.412,E2 -15306.412} C_VEL
LIN {X 0,Y 319.728,Z 305.284,A -85,B 0,C 180,E1 -15310.128,E2 -15310.128} C_VEL
LIN {X 0,Y 319.725,Z 305.283,A -85,B 0,C 180,E1 -15313.993,E2 -15313.993} C_VEL
LIN {X 0,Y 319.652,Z 305.29,A -85,B 0,C 180,E1 -15317.927,E2 -15317.927} C_VEL
LIN {X 0,Y 319.609,Z 305.296,A -85,B 0,C 180,E1 -15320.599,E2 -15320.599} C_VEL
LIN {X 0,Y 319.564,Z 305.304,A -85,B 0,C 180,E1 -15323.32,E2 -15323.32} C_VEL
LIN {X 0,Y 319.628,Z 305.296,A -85,B 0,C 180,E1 -15326.089,E2 -15326.089} C_VEL
LIN {X 0,Y 319.574,Z 305.3,A -85,B 0,C 180,E1 -15328.935,E2 -15328.935} C_VEL
LIN {X 0,Y 319.525,Z 305.306,A -85,B 0,C 180,E1 -15331.863,E2 -15331.863} C_VEL
LIN {X 0,Y 319.575,Z 305.301,A -85,B 0,C 180,E1 -15335.544,E2 -15335.544} C_VEL
LIN {X 0,Y 319.552,Z 305.306,A -85,B 0,C 180,E1 -15338.011,E2 -15338.011} C_VEL
LIN {X 0,Y 319.538,Z 305.429,A -85,B 0,C 180,E1 -15341.287,E2 -15341.287} C_VEL
LIN {X 0,Y 319.954,Z 308.123,A -85,B 0,C 180,E1 -15344.66,E2 -15344.66} C_VEL
LIN {X 0,Y 320.15,Z 310.225,A -85,B 0,C 180,E1 -15347.117,E2 -15347.117} C_VEL
LIN {X 0,Y 320.037,Z 313.274,A -85,B 0,C 180,E1 -15350.445,E2 -15350.445} C_VEL
LIN {X 0,Y 319.742,Z 316.327,A -85,B 0,C 180,E1 -15353.598,E2 -15353.598} C_VEL
LIN {X 0,Y 319.395,Z 319.941,A -85,B 0,C 180,E1 -15357.186,E2 -15357.186} C_VEL
LIN {X 0,Y 320.343,Z 323.046,A -85,B 0,C 180,E1 -15357.402,E2 -15357.402} C_VEL
LIN {X 0,Y 325.98,Z 337.006,A -85,B 0,C 180,E1 -15358.549,E2 -15358.549} C_VEL
LIN {X 0,Y 330.557,Z 351.497,A -85,B 0,C 180,E1 -15359.814,E2 -15359.814} C_VEL
LIN {X 0,Y 333.621,Z 364.135,A -85,B 0,C 180,E1 -15361.02,E2 -15361.02} C_VEL
LIN {X 0,Y 335.317,Z 374.406,A -85,B 0,C 180,E1 -15362.059,E2 -15362.059} C_VEL
LIN {X 0,Y 333.347,Z 387.416,A -85,B 0,C 180,E1 -15363.215,E2 -15363.215} C_VEL
LIN {X 0,Y 331.009,Z 400.901,A -85,B 0,C 180,E1 -15364.705,E2 -15364.705} C_VEL
LIN {X 0,Y 328.667,Z 413.14,A -85,B 0,C 180,E1 -15366.364,E2 -15366.364} C_VEL
LIN {X 0,Y 326.442,Z 424.608,A -85,B 0,C 180,E1 -15368.263,E2 -15368.263} C_VEL
LIN {X 0,Y 324.222,Z 435.125,A -85,B 0,C 180,E1 -15370.368,E2 -15370.368} C_VEL
LIN {X 0,Y 322.332,Z 444.119,A -85,B 0,C 180,E1 -15372.555,E2 -15372.555} C_VEL
LIN {X 0,Y 320.843,Z 451.573,A -85,B 0,C 180,E1 -15374.761,E2 -15374.761} C_VEL
LIN {X 0,Y 319.601,Z 458.542,A -85,B 0,C 180,E1 -15377.298,E2 -15377.298} C_VEL
LIN {X 0,Y 318.688,Z 464.018,A -85,B 0,C 180,E1 -15379.839,E2 -15379.839} C_VEL
LIN {X 0,Y 318.124,Z 468.153,A -85,B 0,C 180,E1 -15382.384,E2 -15382.384} C_VEL
LIN {X 0,Y 317.849,Z 471.058,A -85,B 0,C 180,E1 -15384.926,E2 -15384.926} C_VEL
LIN {X 0,Y 317.754,Z 472.804,A -85,B 0,C 180,E1 -15387.465,E2 -15387.465} C_VEL
LIN {X 0,Y 317.704,Z 473.414,A -85,B 0,C 180,E1 -15390,E2 -15390} C_VEL
LIN {X 0,Y 317.754,Z 472.846,A -85,B 0,C 180,E1 -15392.536,E2 -15392.536} C_VEL
LIN {X 0,Y 317.848,Z 471.156,A -85,B 0,C 180,E1 -15395.075,E2 -15395.075} C_VEL
LIN {X 0,Y 318.124,Z 468.302,A -85,B 0,C 180,E1 -15397.617,E2 -15397.617} C_VEL
LIN {X 0,Y 318.652,Z 464.219,A -85,B 0,C 180,E1 -15400.163,E2 -15400.163} C_VEL
LIN {X 0,Y 319.576,Z 458.805,A -85,B 0,C 180,E1 -15402.704,E2 -15402.704} C_VEL
LIN {X 0,Y 320.775,Z 451.91,A -85,B 0,C 180,E1 -15405.243,E2 -15405.243} C_VEL
LIN {X 0,Y 322.492,Z 443.303,A -85,B 0,C 180,E1 -15407.764,E2 -15407.764} C_VEL
LIN {X 0,Y 324.41,Z 434.154,A -85,B 0,C 180,E1 -15409.951,E2 -15409.951} C_VEL
LIN {X 0,Y 326.582,Z 424.09,A -85,B 0,C 180,E1 -15411.938,E2 -15411.938} C_VEL
LIN {X 0,Y 328.813,Z 412.777,A -85,B 0,C 180,E1 -15413.793,E2 -15413.793} C_VEL
LIN {X 0,Y 331.124,Z 400.464,A -85,B 0,C 180,E1 -15415.455,E2 -15415.455} C_VEL
LIN {X 0,Y 333.238,Z 388.34,A -85,B 0,C 180,E1 -15416.795,E2 -15416.795} C_VEL
LIN {X 0,Y 335.295,Z 375.162,A -85,B 0,C 180,E1 -15417.981,E2 -15417.981} C_VEL
LIN {X 0,Y 335.447,Z 373.965,A -85,B 0,C 180,E1 -15418.083,E2 -15418.083} C_VEL
LIN {X 0,Y 332.907,Z 360.626,A -85,B 0,C 180,E1 -15419.429,E2 -15419.429} C_VEL
LIN {X 0,Y 329.005,Z 346.227,A -85,B 0,C 180,E1 -15420.766,E2 -15420.766} C_VEL
LIN {X 0,Y 324.135,Z 332.138,A -85,B 0,C 180,E1 -15421.97,E2 -15421.97} C_VEL
LIN {X 0,Y 319.562,Z 320.909,A -85,B 0,C 180,E1 -15422.871,E2 -15422.871} C_VEL
LIN {X 0,Y 319.415,Z 319.933,A -85,B 0,C 180,E1 -15422.95,E2 -15422.95} C_VEL
LIN {X 0,Y 319.741,Z 316.464,A -85,B 0,C 180,E1 -15426.403,E2 -15426.403} C_VEL
LIN {X 0,Y 320.069,Z 313.197,A -85,B 0,C 180,E1 -15429.779,E2 -15429.779} C_VEL
LIN {X 0,Y 320.165,Z 310.361,A -85,B 0,C 180,E1 -15432.882,E2 -15432.882} C_VEL
LIN {X 0,Y 319.855,Z 307.327,A -85,B 0,C 180,E1 -15436.476,E2 -15436.476} C_VEL
LIN {X 0,Y 319.566,Z 305.535,A -85,B 0,C 180,E1 -15438.717,E2 -15438.717} C_VEL
LIN {X 0,Y 319.561,Z 305.308,A -85,B 0,C 180,E1 -15442.348,E2 -15442.348} C_VEL
LIN {X 0,Y 319.559,Z 305.309,A -85,B 0,C 180,E1 -15445.123,E2 -15445.123} C_VEL
LIN {X 0,Y 319.559,Z 305.307,A -85,B 0,C 180,E1 -15446.425,E2 -15446.425} C_VEL
LIN {X 0,Y 318.953,Z 305.388,A -85,B 0,C 180,E1 -15447.476,E2 -15447.476} C_VEL
LIN {X 0,Y 316.143,Z 305.742,A -85,B 0,C 180,E1 -15449.187,E2 -15449.187} C_VEL
LIN {X 0,Y 313.703,Z 306.042,A -85,B 0,C 180,E1 -15450.574,E2 -15450.574} C_VEL
LIN {X 0,Y 312.619,Z 306.17,A -85,B 0,C 180,E1 -15451.647,E2 -15451.647} C_VEL
LIN {X 0,Y 312.513,Z 306.181,A -85,B 0,C 180,E1 -15452.011,E2 -15452.011} C_VEL
LIN {X 0,Y 312.547,Z 306.178,A -85,B 0,C 180,E1 -15454.707,E2 -15454.707} C_VEL
LIN {X 0,Y 312.561,Z 306.174,A -85,B 0,C 180,E1 -15457.527,E2 -15457.527} C_VEL
LIN {X 0,Y 312.637,Z 306.167,A -85,B 0,C 180,E1 -15461.656,E2 -15461.656} C_VEL
LIN {X 0,Y 312.692,Z 306.16,A -85,B 0,C 180,E1 -15465.686,E2 -15465.686} C_VEL
LIN {X 0,Y 312.684,Z 306.161,A -85,B 0,C 180,E1 -15469.641,E2 -15469.641} C_VEL
LIN {X 0,Y 312.794,Z 306.148,A -85,B 0,C 180,E1 -15472.252,E2 -15472.252} C_VEL
LIN {X 0,Y 312.702,Z 306.159,A -85,B 0,C 180,E1 -15474.842,E2 -15474.842} C_VEL
LIN {X 0,Y 312.935,Z 306.129,A -85,B 0,C 180,E1 -15477.425,E2 -15477.425} C_VEL
LIN {X 0,Y 313.05,Z 306.116,A -85,B 0,C 180,E1 -15480,E2 -15480} C_VEL
LIN {X 0,Y 312.935,Z 306.13,A -85,B 0,C 180,E1 -15482.574,E2 -15482.574} C_VEL
LIN {X 0,Y 312.841,Z 306.141,A -85,B 0,C 180,E1 -15486.449,E2 -15486.449} C_VEL
LIN {X 0,Y 312.749,Z 306.154,A -85,B 0,C 180,E1 -15489.05,E2 -15489.05} C_VEL
LIN {X 0,Y 312.632,Z 306.168,A -85,B 0,C 180,E1 -15492.991,E2 -15492.991} C_VEL
LIN {X 0,Y 312.636,Z 306.168,A -85,B 0,C 180,E1 -15495.65,E2 -15495.65} C_VEL
LIN {X 0,Y 312.607,Z 306.17,A -85,B 0,C 180,E1 -15499.225,E2 -15499.225} C_VEL
LIN {X 0,Y 312.524,Z 306.182,A -85,B 0,C 180,E1 -15502.78,E2 -15502.78} C_VEL
LIN {X 0,Y 312.6,Z 306.174,A -85,B 0,C 180,E1 -15505.935,E2 -15505.935} C_VEL
LIN {X 0,Y 312.536,Z 306.185,A -85,B 0,C 180,E1 -15509.651,E2 -15509.651} C_VEL
LIN {X 0,Y 312.518,Z 306.191,A -85,B 0,C 180,E1 -15513.689,E2 -15513.689} C_VEL
LIN {X 0,Y 312.524,Z 306.222,A -85,B 0,C 180,E1 -15517.385,E2 -15517.385} C_VEL
LIN {X 0,Y 312.914,Z 308.899,A -85,B 0,C 180,E1 -15520.642,E2 -15520.642} C_VEL
LIN {X 0,Y 313.394,Z 312,A -85,B 0,C 180,E1 -15524.142,E2 -15524.142} C_VEL
LIN {X 0,Y 313.6,Z 313.756,A -85,B 0,C 180,E1 -15525.994,E2 -15525.994} C_VEL
LIN {X 0,Y 313.661,Z 315.487,A -85,B 0,C 180,E1 -15527.764,E2 -15527.764} C_VEL
LIN {X 0,Y 313.367,Z 318.979,A -85,B 0,C 180,E1 -15531.1,E2 -15531.1} C_VEL
LIN {X 0,Y 312.931,Z 322.434,A -85,B 0,C 180,E1 -15534.273,E2 -15534.273} C_VEL
LIN {X 0,Y 312.658,Z 324.745,A -85,B 0,C 180,E1 -15536.31,E2 -15536.31} C_VEL
LIN {X 0,Y 313.641,Z 327.943,A -85,B 0,C 180,E1 -15536.533,E2 -15536.533} C_VEL
LIN {X 0,Y 318.638,Z 340.978,A -85,B 0,C 180,E1 -15537.602,E2 -15537.602} C_VEL
LIN {X 0,Y 322.592,Z 353.515,A -85,B 0,C 180,E1 -15538.71,E2 -15538.71} C_VEL
LIN {X 0,Y 325.937,Z 367.127,A -85,B 0,C 180,E1 -15539.997,E2 -15539.997} C_VEL
LIN {X 0,Y 328.246,Z 380.582,A -85,B 0,C 180,E1 -15541.383,E2 -15541.383} C_VEL
LIN {X 0,Y 328.33,Z 383.279,A -85,B 0,C 180,E1 -15541.656,E2 -15541.656} C_VEL
LIN {X 0,Y 326.125,Z 396.53,A -85,B 0,C 180,E1 -15542.919,E2 -15542.919} C_VEL
LIN {X 0,Y 323.679,Z 409.432,A -85,B 0,C 180,E1 -15544.434,E2 -15544.434} C_VEL
LIN {X 0,Y 321.29,Z 421.243,A -85,B 0,C 180,E1 -15546.129,E2 -15546.129} C_VEL
LIN {X 0,Y 319.017,Z 432.065,A -85,B 0,C 180,E1 -15548.006,E2 -15548.006} C_VEL
LIN {X 0,Y 317.019,Z 441.245,A -85,B 0,C 180,E1 -15549.902,E2 -15549.902} C_VEL
LIN {X 0,Y 315.132,Z 450.25,A -85,B 0,C 180,E1 -15552.142,E2 -15552.142} C_VEL
LIN {X 0,Y 313.422,Z 458.407,A -85,B 0,C 180,E1 -15554.624,E2 -15554.624} C_VEL
LIN {X 0,Y 312.345,Z 464.685,A -85,B 0,C 180,E1 -15556.996,E2 -15556.996} C_VEL
LIN {X 0,Y 311.432,Z 470.161,A -85,B 0,C 180,E1 -15559.599,E2 -15559.599} C_VEL
LIN {X 0,Y 310.948,Z 474.301,A -85,B 0,C 180,E1 -15562.206,E2 -15562.206} C_VEL
LIN {X 0,Y 310.683,Z 477.203,A -85,B 0,C 180,E1 -15564.808,E2 -15564.808} C_VEL
LIN {X 0,Y 310.645,Z 478.933,A -85,B 0,C 180,E1 -15567.406,E2 -15567.406} C_VEL
LIN {X 0,Y 310.615,Z 479.525,A -85,B 0,C 180,E1 -15569.999,E2 -15569.999} C_VEL
LIN {X 0,Y 310.645,Z 478.925,A -85,B 0,C 180,E1 -15572.593,E2 -15572.593} C_VEL
LIN {X 0,Y 310.688,Z 477.184,A -85,B 0,C 180,E1 -15575.191,E2 -15575.191} C_VEL
LIN {X 0,Y 310.948,Z 474.276,A -85,B 0,C 180,E1 -15577.793,E2 -15577.793} C_VEL
LIN {X 0,Y 311.431,Z 470.133,A -85,B 0,C 180,E1 -15580.4,E2 -15580.4} C_VEL
LIN {X 0,Y 312.343,Z 464.643,A -85,B 0,C 180,E1 -15583.003,E2 -15583.003} C_VEL
LIN {X 0,Y 313.555,Z 457.657,A -85,B 0,C 180,E1 -15585.602,E2 -15585.602} C_VEL
LIN {X 0,Y 315.361,Z 448.965,A -85,B 0,C 180,E1 -15588.179,E2 -15588.179} C_VEL
LIN {X 0,Y 317.383,Z 439.73,A -85,B 0,C 180,E1 -15590.411,E2 -15590.411} C_VEL
LIN {X 0,Y 319.36,Z 430.347,A -85,B 0,C 180,E1 -15592.307,E2 -15592.307} C_VEL
LIN {X 0,Y 321.905,Z 418.159,A -85,B 0,C 180,E1 -15594.335,E2 -15594.335} C_VEL
LIN {X 0,Y 324.372,Z 405.734,A -85,B 0,C 180,E1 -15596.023,E2 -15596.023} C_VEL
LIN {X 0,Y 326.881,Z 391.983,A -85,B 0,C 180,E1 -15597.532,E2 -15597.532} C_VEL
LIN {X 0,Y 328.381,Z 382.142,A -85,B 0,C 180,E1 -15598.428,E2 -15598.428} C_VEL
LIN {X 0,Y 326.149,Z 368.503,A -85,B 0,C 180,E1 -15599.851,E2 -15599.851} C_VEL
LIN {X 0,Y 322.67,Z 354.002,A -85,B 0,C 180,E1 -15601.229,E2 -15601.229} C_VEL
LIN {X 0,Y 319.004,Z 342.073,A -85,B 0,C 180,E1 -15602.28,E2 -15602.28} C_VEL
LIN {X 0,Y 313.696,Z 328.11,A -85,B 0,C 180,E1 -15603.427,E2 -15603.427} C_VEL
LIN {X 0,Y 312.63,Z 324.748,A -85,B 0,C 180,E1 -15603.683,E2 -15603.683} C_VEL
LIN {X 0,Y 313.13,Z 320.704,A -85,B 0,C 180,E1 -15607.299,E2 -15607.299} C_VEL
LIN {X 0,Y 313.526,Z 317.225,A -85,B 0,C 180,E1 -15610.545,E2 -15610.545} C_VEL
LIN {X 0,Y 313.637,Z 315.413,A -85,B 0,C 180,E1 -15612.314,E2 -15612.314} C_VEL
LIN {X 0,Y 313.583,Z 313.584,A -85,B 0,C 180,E1 -15614.178,E2 -15614.178} C_VEL
LIN {X 0,Y 313.139,Z 310.257,A -85,B 0,C 180,E1 -15617.784,E2 -15617.784} C_VEL
LIN {X 0,Y 312.602,Z 306.761,A -85,B 0,C 180,E1 -15621.893,E2 -15621.893} C_VEL
LIN {X 0,Y 312.521,Z 306.185,A -85,B 0,C 180,E1 -15622.614,E2 -15622.614} C_VEL
LIN {X 0,Y 312.513,Z 306.189,A -85,B 0,C 180,E1 -15626.311,E2 -15626.311} C_VEL
LIN {X 0,Y 312.532,Z 306.186,A -85,B 0,C 180,E1 -15630.349,E2 -15630.349} C_VEL
LIN {X 0,Y 312.596,Z 306.174,A -85,B 0,C 180,E1 -15634.064,E2 -15634.064} C_VEL
LIN {X 0,Y 312.581,Z 306.174,A -85,B 0,C 180,E1 -15637.529,E2 -15637.529} C_VEL
LIN {X 0,Y 312.632,Z 306.169,A -85,B 0,C 180,E1 -15641.656,E2 -15641.656} C_VEL
LIN {X 0,Y 312.687,Z 306.158,A -85,B 0,C 180,E1 -15645.686,E2 -15645.686} C_VEL
LIN {X 0,Y 312.678,Z 306.162,A -85,B 0,C 180,E1 -15649.641,E2 -15649.641} C_VEL
LIN {X 0,Y 312.789,Z 306.148,A -85,B 0,C 180,E1 -15652.252,E2 -15652.252} C_VEL
LIN {X 0,Y 312.699,Z 306.156,A -85,B 0,C 180,E1 -15654.842,E2 -15654.842} C_VEL
LIN {X 0,Y 312.931,Z 306.125,A -85,B 0,C 180,E1 -15657.426,E2 -15657.426} C_VEL
LIN {X 0,Y 313.06,Z 306.115,A -85,B 0,C 180,E1 -15660,E2 -15660} C_VEL
LIN {X 0,Y 312.931,Z 306.13,A -85,B 0,C 180,E1 -15662.575,E2 -15662.575} C_VEL
LIN {X 0,Y 312.836,Z 306.143,A -85,B 0,C 180,E1 -15666.45,E2 -15666.45} C_VEL
LIN {X 0,Y 312.743,Z 306.151,A -85,B 0,C 180,E1 -15669.051,E2 -15669.051} C_VEL
LIN {X 0,Y 312.628,Z 306.168,A -85,B 0,C 180,E1 -15672.992,E2 -15672.992} C_VEL
LIN {X 0,Y 312.632,Z 306.168,A -85,B 0,C 180,E1 -15675.65,E2 -15675.65} C_VEL
LIN {X 0,Y 312.624,Z 306.169,A -85,B 0,C 180,E1 -15679.237,E2 -15679.237} C_VEL
LIN {X 0,Y 312.54,Z 306.18,A -85,B 0,C 180,E1 -15682.79,E2 -15682.79} C_VEL
LIN {X 0,Y 312.597,Z 306.172,A -85,B 0,C 180,E1 -15685.936,E2 -15685.936} C_VEL
LIN {X 0,Y 312.532,Z 306.176,A -85,B 0,C 180,E1 -15689.651,E2 -15689.651} C_VEL
LIN {X 0,Y 312.514,Z 306.179,A -85,B 0,C 180,E1 -15693.69,E2 -15693.69} C_VEL
LIN {X 0,Y 312.521,Z 306.181,A -85,B 0,C 180,E1 -15697.386,E2 -15697.386} C_VEL
LIN {X 0,Y 312.47,Z 306.204,A -85,B 0,C 180,E1 -15700.712,E2 -15700.712} C_VEL
LIN {X 0,Y 312.88,Z 308.849,A -85,B 0,C 180,E1 -15704.133,E2 -15704.133} C_VEL
LIN {X 0,Y 313.065,Z 310.318,A -85,B 0,C 180,E1 -15705.92,E2 -15705.92} C_VEL
LIN {X 0,Y 313.141,Z 311.923,A -85,B 0,C 180,E1 -15707.786,E2 -15707.786} C_VEL
LIN {X 0,Y 312.929,Z 314.879,A -85,B 0,C 180,E1 -15711.036,E2 -15711.036} C_VEL
LIN {X 0,Y 312.662,Z 317.929,A -85,B 0,C 180,E1 -15714.239,E2 -15714.239} C_VEL
LIN {X 0,Y 312.402,Z 320.008,A -85,B 0,C 180,E1 -15716.344,E2 -15716.344} C_VEL
LIN {X 0,Y 313.542,Z 323.354,A -85,B 0,C 180,E1 -15716.61,E2 -15716.61} C_VEL
LIN {X 0,Y 319.394,Z 337.815,A -85,B 0,C 180,E1 -15717.86,E2 -15717.86} C_VEL
LIN {X 0,Y 323.714,Z 351.267,A -85,B 0,C 180,E1 -15719.086,E2 -15719.086} C_VEL
LIN {X 0,Y 327.143,Z 365.163,A -85,B 0,C 180,E1 -15720.465,E2 -15720.465} C_VEL
LIN {X 0,Y 328.883,Z 375.601,A -85,B 0,C 180,E1 -15721.573,E2 -15721.573} C_VEL
LIN {X 0,Y 326.757,Z 388.92,A -85,B 0,C 180,E1 -15722.804,E2 -15722.804} C_VEL
LIN {X 0,Y 324.355,Z 402.145,A -85,B 0,C 180,E1 -15724.321,E2 -15724.321} C_VEL
LIN {X 0,Y 322.158,Z 413.213,A -85,B 0,C 180,E1 -15725.857,E2 -15725.857} C_VEL
LIN {X 0,Y 319.802,Z 424.806,A -85,B 0,C 180,E1 -15727.814,E2 -15727.814} C_VEL
LIN {X 0,Y 317.482,Z 435.197,A -85,B 0,C 180,E1 -15729.934,E2 -15729.934} C_VEL
LIN {X 0,Y 315.512,Z 444.191,A -85,B 0,C 180,E1 -15732.166,E2 -15732.166} C_VEL
LIN {X 0,Y 313.931,Z 451.645,A -85,B 0,C 180,E1 -15734.417,E2 -15734.417} C_VEL
LIN {X 0,Y 312.653,Z 458.612,A -85,B 0,C 180,E1 -15737.01,E2 -15737.01} C_VEL
LIN {X 0,Y 311.645,Z 464.089,A -85,B 0,C 180,E1 -15739.607,E2 -15739.607} C_VEL
LIN {X 0,Y 311.053,Z 468.223,A -85,B 0,C 180,E1 -15742.209,E2 -15742.209} C_VEL
LIN {X 0,Y 310.772,Z 471.127,A -85,B 0,C 180,E1 -15744.811,E2 -15744.811} C_VEL
LIN {X 0,Y 310.678,Z 472.873,A -85,B 0,C 180,E1 -15747.407,E2 -15747.407} C_VEL
LIN {X 0,Y 310.617,Z 473.483,A -85,B 0,C 180,E1 -15750.001,E2 -15750.001} C_VEL
LIN {X 0,Y 310.678,Z 472.915,A -85,B 0,C 180,E1 -15752.594,E2 -15752.594} C_VEL
LIN {X 0,Y 310.772,Z 471.224,A -85,B 0,C 180,E1 -15755.19,E2 -15755.19} C_VEL
LIN {X 0,Y 311.052,Z 468.371,A -85,B 0,C 180,E1 -15757.792,E2 -15757.792} C_VEL
LIN {X 0,Y 311.615,Z 464.287,A -85,B 0,C 180,E1 -15760.395,E2 -15760.395} C_VEL
LIN {X 0,Y 312.625,Z 458.873,A -85,B 0,C 180,E1 -15762.992,E2 -15762.992} C_VEL
LIN {X 0,Y 313.876,Z 451.978,A -85,B 0,C 180,E1 -15765.587,E2 -15765.587} C_VEL
LIN {X 0,Y 315.695,Z 443.37,A -85,B 0,C 180,E1 -15768.16,E2 -15768.16} C_VEL
LIN {X 0,Y 317.678,Z 434.221,A -85,B 0,C 180,E1 -15770.392,E2 -15770.392} C_VEL
LIN {X 0,Y 319.898,Z 424.461,A -85,B 0,C 180,E1 -15772.361,E2 -15772.361} C_VEL
LIN {X 0,Y 322.286,Z 412.843,A -85,B 0,C 180,E1 -15774.306,E2 -15774.306} C_VEL
LIN {X 0,Y 324.676,Z 400.529,A -85,B 0,C 180,E1 -15775.998,E2 -15775.998} C_VEL
LIN {X 0,Y 326.917,Z 388.404,A -85,B 0,C 180,E1 -15777.356,E2 -15777.356} C_VEL
LIN {X 0,Y 328.938,Z 375.226,A -85,B 0,C 180,E1 -15778.571,E2 -15778.571} C_VEL
LIN {X 0,Y 326.494,Z 362.09,A -85,B 0,C 180,E1 -15779.956,E2 -15779.956} C_VEL
LIN {X 0,Y 322.586,Z 347.463,A -85,B 0,C 180,E1 -15781.377,E2 -15781.377} C_VEL
LIN {X 0,Y 317.85,Z 333.727,A -85,B 0,C 180,E1 -15782.617,E2 -15782.617} C_VEL
LIN {X 0,Y 313.366,Z 323.07,A -85,B 0,C 180,E1 -15783.539,E2 -15783.539} C_VEL
LIN {X 0,Y 312.435,Z 320.006,A -85,B 0,C 180,E1 -15783.786,E2 -15783.786} C_VEL
LIN {X 0,Y 312.803,Z 316.53,A -85,B 0,C 180,E1 -15787.346,E2 -15787.346} C_VEL
LIN {X 0,Y 313.099,Z 313.474,A -85,B 0,C 180,E1 -15790.613,E2 -15790.613} C_VEL
LIN {X 0,Y 313.167,Z 311.962,A -85,B 0,C 180,E1 -15792.318,E2 -15792.318} C_VEL
LIN {X 0,Y 312.904,Z 308.917,A -85,B 0,C 180,E1 -15795.95,E2 -15795.95} C_VEL
LIN {X 0,Y 312.511,Z 306.305,A -85,B 0,C 180,E1 -15799.294,E2 -15799.294} C_VEL
LIN {X 0,Y 312.525,Z 306.185,A -85,B 0,C 180,E1 -15802.615,E2 -15802.615} C_VEL
LIN {X 0,Y 312.513,Z 306.184,A -85,B 0,C 180,E1 -15806.411,E2 -15806.411} C_VEL
LIN {X 0,Y 312.495,Z 306.186,A -85,B 0,C 180,E1 -15810.345,E2 -15810.345} C_VEL
LIN {X 0,Y 312.513,Z 306.181,A -85,B 0,C 180,E1 -15812.011,E2 -15812.011} C_VEL
LIN {X 0,Y 311.801,Z 306.269,A -85,B 0,C 180,E1 -15813.087,E2 -15813.087} C_VEL
LIN {X 0,Y 308.947,Z 306.626,A -85,B 0,C 180,E1 -15814.839,E2 -15814.839} C_VEL
LIN {X 0,Y 306.56,Z 306.924,A -85,B 0,C 180,E1 -15816.259,E2 -15816.259} C_VEL
LIN {X 0,Y 305.542,Z 307.049,A -85,B 0,C 180,E1 -15817.358,E2 -15817.358} C_VEL
LIN {X 0,Y 305.461,Z 307.057,A -85,B 0,C 180,E1 -15817.731,E2 -15817.731} C_VEL
LIN {X 0,Y 305.588,Z 307.042,A -85,B 0,C 180,E1 -15821.217,E2 -15821.217} C_VEL
LIN {X 0,Y 305.647,Z 307.038,A -85,B 0,C 180,E1 -15825.349,E2 -15825.349} C_VEL
LIN {X 0,Y 305.622,Z 307.041,A -85,B 0,C 180,E1 -15829.399,E2 -15829.399} C_VEL
LIN {X 0,Y 305.745,Z 307.025,A -85,B 0,C 180,E1 -15832.072,E2 -15832.072} C_VEL
LIN {X 0,Y 305.67,Z 307.035,A -85,B 0,C 180,E1 -15834.723,E2 -15834.723} C_VEL
LIN {X 0,Y 305.952,Z 307,A -85,B 0,C 180,E1 -15838.684,E2 -15838.684} C_VEL
LIN {X 0,Y 305.95,Z 307,A -85,B 0,C 180,E1 -15841.316,E2 -15841.316} C_VEL
LIN {X 0,Y 305.671,Z 307.034,A -85,B 0,C 180,E1 -15845.277,E2 -15845.277} C_VEL
LIN {X 0,Y 305.745,Z 307.027,A -85,B 0,C 180,E1 -15847.927,E2 -15847.927} C_VEL
LIN {X 0,Y 305.597,Z 307.046,A -85,B 0,C 180,E1 -15851.945,E2 -15851.945} C_VEL
LIN {X 0,Y 305.636,Z 307.041,A -85,B 0,C 180,E1 -15855.035,E2 -15855.035} C_VEL
LIN {X 0,Y 305.578,Z 307.047,A -85,B 0,C 180,E1 -15858.783,E2 -15858.783} C_VEL
LIN {X 0,Y 305.485,Z 307.06,A -85,B 0,C 180,E1 -15863.039,E2 -15863.039} C_VEL
LIN {X 0,Y 305.53,Z 307.054,A -85,B 0,C 180,E1 -15866.221,E2 -15866.221} C_VEL
LIN {X 0,Y 305.486,Z 307.062,A -85,B 0,C 180,E1 -15869.047,E2 -15869.047} C_VEL
LIN {X 0,Y 305.44,Z 307.071,A -85,B 0,C 180,E1 -15871.952,E2 -15871.952} C_VEL
LIN {X 0,Y 305.461,Z 307.07,A -85,B 0,C 180,E1 -15875.113,E2 -15875.113} C_VEL
LIN {X 0,Y 305.458,Z 307.07,A -85,B 0,C 180,E1 -15876.742,E2 -15876.742} C_VEL
LIN {X 0,Y 305.847,Z 309.656,A -85,B 0,C 180,E1 -15880.046,E2 -15880.046} C_VEL
LIN {X 0,Y 306.272,Z 312.623,A -85,B 0,C 180,E1 -15883.504,E2 -15883.504} C_VEL
LIN {X 0,Y 306.585,Z 315.418,A -85,B 0,C 180,E1 -15886.551,E2 -15886.551} C_VEL
LIN {X 0,Y 306.509,Z 318.002,A -85,B 0,C 180,E1 -15889.171,E2 -15889.171} C_VEL
LIN {X 0,Y 306.27,Z 320.641,A -85,B 0,C 180,E1 -15891.715,E2 -15891.715} C_VEL
LIN {X 0,Y 305.686,Z 324.657,A -85,B 0,C 180,E1 -15895.423,E2 -15895.423} C_VEL
LIN {X 0,Y 306.787,Z 328.053,A -85,B 0,C 180,E1 -15895.688,E2 -15895.688} C_VEL
LIN {X 0,Y 311.14,Z 338.893,A -85,B 0,C 180,E1 -15896.636,E2 -15896.636} C_VEL
LIN {X 0,Y 315.92,Z 353.535,A -85,B 0,C 180,E1 -15897.977,E2 -15897.977} C_VEL
LIN {X 0,Y 319.271,Z 367.312,A -85,B 0,C 180,E1 -15899.324,E2 -15899.324} C_VEL
LIN {X 0,Y 321.551,Z 380.441,A -85,B 0,C 180,E1 -15900.723,E2 -15900.723} C_VEL
LIN {X 0,Y 321.905,Z 384.484,A -85,B 0,C 180,E1 -15901.166,E2 -15901.166} C_VEL
LIN {X 0,Y 319.505,Z 397.891,A -85,B 0,C 180,E1 -15902.488,E2 -15902.488} C_VEL
LIN {X 0,Y 317.012,Z 410.54,A -85,B 0,C 180,E1 -15904.033,E2 -15904.033} C_VEL
LIN {X 0,Y 314.775,Z 421.177,A -85,B 0,C 180,E1 -15905.603,E2 -15905.603} C_VEL
LIN {X 0,Y 312.366,Z 431.998,A -85,B 0,C 180,E1 -15907.512,E2 -15907.512} C_VEL
LIN {X 0,Y 310.319,Z 441.178,A -85,B 0,C 180,E1 -15909.449,E2 -15909.449} C_VEL
LIN {X 0,Y 308.321,Z 450.182,A -85,B 0,C 180,E1 -15911.734,E2 -15911.734} C_VEL
LIN {X 0,Y 306.658,Z 457.649,A -85,B 0,C 180,E1 -15914.037,E2 -15914.037} C_VEL
LIN {X 0,Y 305.379,Z 464.616,A -85,B 0,C 180,E1 -15916.694,E2 -15916.694} C_VEL
LIN {X 0,Y 304.398,Z 470.092,A -85,B 0,C 180,E1 -15919.356,E2 -15919.356} C_VEL
LIN {X 0,Y 303.868,Z 474.232,A -85,B 0,C 180,E1 -15922.023,E2 -15922.023} C_VEL
LIN {X 0,Y 303.596,Z 477.134,A -85,B 0,C 180,E1 -15924.687,E2 -15924.687} C_VEL
LIN {X 0,Y 303.571,Z 478.865,A -85,B 0,C 180,E1 -15927.346,E2 -15927.346} C_VEL
LIN {X 0,Y 303.531,Z 479.456,A -85,B 0,C 180,E1 -15929.999,E2 -15929.999} C_VEL
LIN {X 0,Y 303.571,Z 478.856,A -85,B 0,C 180,E1 -15932.653,E2 -15932.653} C_VEL
LIN {X 0,Y 303.623,Z 476.918,A -85,B 0,C 180,E1 -15935.544,E2 -15935.544} C_VEL
LIN {X 0,Y 303.868,Z 474.206,A -85,B 0,C 180,E1 -15937.976,E2 -15937.976} C_VEL
LIN {X 0,Y 304.396,Z 470.062,A -85,B 0,C 180,E1 -15940.643,E2 -15940.643} C_VEL
LIN {X 0,Y 305.378,Z 464.572,A -85,B 0,C 180,E1 -15943.305,E2 -15943.305} C_VEL
LIN {X 0,Y 306.658,Z 457.586,A -85,B 0,C 180,E1 -15945.962,E2 -15945.962} C_VEL
LIN {X 0,Y 308.563,Z 448.893,A -85,B 0,C 180,E1 -15948.594,E2 -15948.594} C_VEL
LIN {X 0,Y 310.702,Z 439.658,A -85,B 0,C 180,E1 -15950.87,E2 -15950.87} C_VEL
LIN {X 0,Y 313.036,Z 429.174,A -85,B 0,C 180,E1 -15953.002,E2 -15953.002} C_VEL
LIN {X 0,Y 315.4,Z 418.086,A -85,B 0,C 180,E1 -15954.871,E2 -15954.871} C_VEL
LIN {X 0,Y 317.993,Z 405.661,A -85,B 0,C 180,E1 -15956.585,E2 -15956.585} C_VEL
LIN {X 0,Y 320.56,Z 391.99,A -85,B 0,C 180,E1 -15958.113,E2 -15958.113} C_VEL
LIN {X 0,Y 321.945,Z 383.718,A -85,B 0,C 180,E1 -15958.883,E2 -15958.883} C_VEL
LIN {X 0,Y 319.829,Z 370.23,A -85,B 0,C 180,E1 -15960.357,E2 -15960.357} C_VEL
LIN {X 0,Y 316.392,Z 355.46,A -85,B 0,C 180,E1 -15961.826,E2 -15961.826} C_VEL
LIN {X 0,Y 311.755,Z 340.747,A -85,B 0,C 180,E1 -15963.183,E2 -15963.183} C_VEL
LIN {X 0,Y 306.973,Z 328.441,A -85,B 0,C 180,E1 -15964.245,E2 -15964.245} C_VEL
LIN {X 0,Y 305.793,Z 325.482,A -85,B 0,C 180,E1 -15964.49,E2 -15964.49} C_VEL
LIN {X 0,Y 305.673,Z 324.65,A -85,B 0,C 180,E1 -15964.572,E2 -15964.572} C_VEL
LIN {X 0,Y 306.242,Z 320.621,A -85,B 0,C 180,E1 -15968.288,E2 -15968.288} C_VEL
LIN {X 0,Y 306.571,Z 317.147,A -85,B 0,C 180,E1 -15971.666,E2 -15971.666} C_VEL
LIN {X 0,Y 306.489,Z 314.243,A -85,B 0,C 180,E1 -15974.696,E2 -15974.696} C_VEL
LIN {X 0,Y 306.057,Z 311.08,A -85,B 0,C 180,E1 -15978.247,E2 -15978.247} C_VEL
LIN {X 0,Y 305.646,Z 308.266,A -85,B 0,C 180,E1 -15981.623,E2 -15981.623} C_VEL
LIN {X 0,Y 305.47,Z 307.064,A -85,B 0,C 180,E1 -15983.26,E2 -15983.26} C_VEL
LIN {X 0,Y 305.459,Z 307.069,A -85,B 0,C 180,E1 -15986.483,E2 -15986.483} C_VEL
LIN {X 0,Y 305.452,Z 307.069,A -85,B 0,C 180,E1 -15989.59,E2 -15989.59} C_VEL
LIN {X 0,Y 305.512,Z 307.058,A -85,B 0,C 180,E1 -15992.608,E2 -15992.608} C_VEL
LIN {X 0,Y 305.501,Z 307.059,A -85,B 0,C 180,E1 -15995.538,E2 -15995.538} C_VEL
LIN {X 0,Y 305.514,Z 307.055,A -85,B 0,C 180,E1 -15999.815,E2 -15999.815} C_VEL
LIN {X 0,Y 305.567,Z 307.045,A -85,B 0,C 180,E1 -16002.603,E2 -16002.603} C_VEL
LIN {X 0,Y 305.642,Z 307.035,A -85,B 0,C 180,E1 -16005.349,E2 -16005.349} C_VEL
LIN {X 0,Y 305.617,Z 307.043,A -85,B 0,C 180,E1 -16009.399,E2 -16009.399} C_VEL
LIN {X 0,Y 305.739,Z 307.025,A -85,B 0,C 180,E1 -16012.073,E2 -16012.073} C_VEL
LIN {X 0,Y 305.667,Z 307.031,A -85,B 0,C 180,E1 -16014.723,E2 -16014.723} C_VEL
LIN {X 0,Y 305.947,Z 307,A -85,B 0,C 180,E1 -16018.684,E2 -16018.684} C_VEL
LIN {X 0,Y 305.947,Z 307.002,A -85,B 0,C 180,E1 -16021.316,E2 -16021.316} C_VEL
LIN {X 0,Y 305.667,Z 307.035,A -85,B 0,C 180,E1 -16025.277,E2 -16025.277} C_VEL
LIN {X 0,Y 305.739,Z 307.021,A -85,B 0,C 180,E1 -16027.928,E2 -16027.928} C_VEL
LIN {X 0,Y 305.592,Z 307.04,A -85,B 0,C 180,E1 -16031.946,E2 -16031.946} C_VEL
LIN {X 0,Y 305.631,Z 307.036,A -85,B 0,C 180,E1 -16035.035,E2 -16035.035} C_VEL
LIN {X 0,Y 305.571,Z 307.048,A -85,B 0,C 180,E1 -16039.446,E2 -16039.446} C_VEL
LIN {X 0,Y 305.485,Z 307.059,A -85,B 0,C 180,E1 -16043.042,E2 -16043.042} C_VEL
LIN {X 0,Y 305.526,Z 307.052,A -85,B 0,C 180,E1 -16046.221,E2 -16046.221} C_VEL
LIN {X 0,Y 305.483,Z 307.055,A -85,B 0,C 180,E1 -16049.048,E2 -16049.048} C_VEL
LIN {X 0,Y 305.437,Z 307.06,A -85,B 0,C 180,E1 -16051.953,E2 -16051.953} C_VEL
LIN {X 0,Y 305.457,Z 307.059,A -85,B 0,C 180,E1 -16055.114,E2 -16055.114} C_VEL
LIN {X 0,Y 305.445,Z 307.064,A -85,B 0,C 180,E1 -16058.53,E2 -16058.53} C_VEL
LIN {X 0,Y 305.457,Z 307.063,A -85,B 0,C 180,E1 -16060.108,E2 -16060.108} C_VEL
LIN {X 0,Y 305.798,Z 309.59,A -85,B 0,C 180,E1 -16063.589,E2 -16063.589} C_VEL
LIN {X 0,Y 306.046,Z 311.902,A -85,B 0,C 180,E1 -16066.457,E2 -16066.457} C_VEL
LIN {X 0,Y 306.089,Z 314.308,A -85,B 0,C 180,E1 -16069.262,E2 -16069.262} C_VEL
LIN {X 0,Y 305.712,Z 318.004,A -85,B 0,C 180,E1 -16073.295,E2 -16073.295} C_VEL
LIN {X 0,Y 305.451,Z 320.088,A -85,B 0,C 180,E1 -16075.474,E2 -16075.474} C_VEL
LIN {X 0,Y 306.622,Z 323.517,A -85,B 0,C 180,E1 -16075.756,E2 -16075.756} C_VEL
LIN {X 0,Y 311.714,Z 335.699,A -85,B 0,C 180,E1 -16076.858,E2 -16076.858} C_VEL
LIN {X 0,Y 316.174,Z 348.686,A -85,B 0,C 180,E1 -16078.099,E2 -16078.099} C_VEL
LIN {X 0,Y 319.963,Z 363.069,A -85,B 0,C 180,E1 -16079.557,E2 -16079.557} C_VEL
LIN {X 0,Y 322.412,Z 376.382,A -85,B 0,C 180,E1 -16081.02,E2 -16081.02} C_VEL
LIN {X 0,Y 320.452,Z 388.994,A -85,B 0,C 180,E1 -16082.223,E2 -16082.223} C_VEL
LIN {X 0,Y 318.153,Z 401.048,A -85,B 0,C 180,E1 -16083.606,E2 -16083.606} C_VEL
LIN {X 0,Y 315.648,Z 413.286,A -85,B 0,C 180,E1 -16085.326,E2 -16085.326} C_VEL
LIN {X 0,Y 313.189,Z 425.004,A -85,B 0,C 180,E1 -16087.346,E2 -16087.346} C_VEL
LIN {X 0,Y 310.769,Z 435.269,A -85,B 0,C 180,E1 -16089.481,E2 -16089.481} C_VEL
LIN {X 0,Y 308.717,Z 444.262,A -85,B 0,C 180,E1 -16091.759,E2 -16091.759} C_VEL
LIN {X 0,Y 307.053,Z 451.716,A -85,B 0,C 180,E1 -16094.059,E2 -16094.059} C_VEL
LIN {X 0,Y 305.681,Z 458.683,A -85,B 0,C 180,E1 -16096.709,E2 -16096.709} C_VEL
LIN {X 0,Y 304.622,Z 464.16,A -85,B 0,C 180,E1 -16099.365,E2 -16099.365} C_VEL
LIN {X 0,Y 304.005,Z 468.293,A -85,B 0,C 180,E1 -16102.028,E2 -16102.028} C_VEL
LIN {X 0,Y 303.686,Z 471.197,A -85,B 0,C 180,E1 -16104.689,E2 -16104.689} C_VEL
LIN {X 0,Y 303.604,Z 472.943,A -85,B 0,C 180,E1 -16107.347,E2 -16107.347} C_VEL
LIN {X 0,Y 303.533,Z 473.552,A -85,B 0,C 180,E1 -16110.001,E2 -16110.001} C_VEL
LIN {X 0,Y 303.604,Z 472.984,A -85,B 0,C 180,E1 -16112.654,E2 -16112.654} C_VEL
LIN {X 0,Y 303.686,Z 471.293,A -85,B 0,C 180,E1 -16115.312,E2 -16115.312} C_VEL
LIN {X 0,Y 304.004,Z 468.439,A -85,B 0,C 180,E1 -16117.974,E2 -16117.974} C_VEL
LIN {X 0,Y 304.597,Z 464.356,A -85,B 0,C 180,E1 -16120.637,E2 -16120.637} C_VEL
LIN {X 0,Y 305.651,Z 458.941,A -85,B 0,C 180,E1 -16123.294,E2 -16123.294} C_VEL
LIN {X 0,Y 306.989,Z 452.045,A -85,B 0,C 180,E1 -16125.946,E2 -16125.946} C_VEL
LIN {X 0,Y 308.915,Z 443.438,A -85,B 0,C 180,E1 -16128.573,E2 -16128.573} C_VEL
LIN {X 0,Y 311,Z 434.288,A -85,B 0,C 180,E1 -16130.85,E2 -16130.85} C_VEL
LIN {X 0,Y 313.181,Z 425.073,A -85,B 0,C 180,E1 -16132.752,E2 -16132.752} C_VEL
LIN {X 0,Y 315.578,Z 413.9,A -85,B 0,C 180,E1 -16134.681,E2 -16134.681} C_VEL
LIN {X 0,Y 318.053,Z 401.779,A -85,B 0,C 180,E1 -16136.404,E2 -16136.404} C_VEL
LIN {X 0,Y 320.34,Z 389.892,A -85,B 0,C 180,E1 -16137.788,E2 -16137.788} C_VEL
LIN {X 0,Y 322.483,Z 377.332,A -85,B 0,C 180,E1 -16138.991,E2 -16138.991} C_VEL
LIN {X 0,Y 320.588,Z 365.702,A -85,B 0,C 180,E1 -16140.279,E2 -16140.279} C_VEL
LIN {X 0,Y 316.903,Z 351.029,A -85,B 0,C 180,E1 -16141.79,E2 -16141.79} C_VEL
LIN {X 0,Y 312.174,Z 336.794,A -85,B 0,C 180,E1 -16143.153,E2 -16143.153} C_VEL
LIN {X 0,Y 306.677,Z 323.58,A -85,B 0,C 180,E1 -16144.356,E2 -16144.356} C_VEL
LIN {X 0,Y 305.54,Z 320.673,A -85,B 0,C 180,E1 -16144.597,E2 -16144.597} C_VEL
LIN {X 0,Y 305.481,Z 320.093,A -85,B 0,C 180,E1 -16144.651,E2 -16144.651} C_VEL
LIN {X 0,Y 305.887,Z 316.334,A -85,B 0,C 180,E1 -16148.631,E2 -16148.631} C_VEL
LIN {X 0,Y 306.121,Z 313.564,A -85,B 0,C 180,E1 -16151.743,E2 -16151.743} C_VEL
LIN {X 0,Y 305.941,Z 310.508,A -85,B 0,C 180,E1 -16155.408,E2 -16155.408} C_VEL
LIN {X 0,Y 305.519,Z 307.457,A -85,B 0,C 180,E1 -16159.386,E2 -16159.386} C_VEL
LIN {X 0,Y 305.448,Z 307.09,A -85,B 0,C 180,E1 -16159.89,E2 -16159.89} C_VEL
LIN {X 0,Y 305.481,Z 307.062,A -85,B 0,C 180,E1 -16163.631,E2 -16163.631} C_VEL
LIN {X 0,Y 305.464,Z 307.063,A -85,B 0,C 180,E1 -16166.483,E2 -16166.483} C_VEL
LIN {X 0,Y 305.429,Z 307.065,A -85,B 0,C 180,E1 -16169.587,E2 -16169.587} C_VEL
LIN {X 0,Y 305.457,Z 307.062,A -85,B 0,C 180,E1 -16172.602,E2 -16172.602} C_VEL
LIN {X 0,Y 305.474,Z 307.058,A -85,B 0,C 180,E1 -16175.536,E2 -16175.536} C_VEL
LIN {X 0,Y 305.461,Z 307.057,A -85,B 0,C 180,E1 -16177.731,E2 -16177.731} C_VEL
LIN {X 0,Y 304.797,Z 307.144,A -85,B 0,C 180,E1 -16178.832,E2 -16178.832} C_VEL
LIN {X 0,Y 301.957,Z 307.493,A -85,B 0,C 180,E1 -16180.625,E2 -16180.625} C_VEL
LIN {X 0,Y 299.579,Z 307.794,A -85,B 0,C 180,E1 -16182.079,E2 -16182.079} C_VEL
LIN {X 0,Y 298.603,Z 307.912,A -85,B 0,C 180,E1 -16183.205,E2 -16183.205} C_VEL
LIN {X 0,Y 298.547,Z 307.918,A -85,B 0,C 180,E1 -16183.586,E2 -16183.586} C_VEL
LIN {X 0,Y 298.55,Z 307.918,A -85,B 0,C 180,E1 -16186.384,E2 -16186.384} C_VEL
LIN {X 0,Y 298.706,Z 307.902,A -85,B 0,C 180,E1 -16191.18,E2 -16191.18} C_VEL
LIN {X 0,Y 298.639,Z 307.911,A -85,B 0,C 180,E1 -16194.598,E2 -16194.598} C_VEL
LIN {X 0,Y 298.919,Z 307.877,A -85,B 0,C 180,E1 -16198.653,E2 -16198.653} C_VEL
LIN {X 0,Y 298.917,Z 307.876,A -85,B 0,C 180,E1 -16201.347,E2 -16201.347} C_VEL
LIN {X 0,Y 298.639,Z 307.91,A -85,B 0,C 180,E1 -16205.401,E2 -16205.401} C_VEL
LIN {X 0,Y 298.706,Z 307.902,A -85,B 0,C 180,E1 -16208.82,E2 -16208.82} C_VEL
LIN {X 0,Y 298.55,Z 307.924,A -85,B 0,C 180,E1 -16213.615,E2 -16213.615} C_VEL
LIN {X 0,Y 298.547,Z 307.923,A -85,B 0,C 180,E1 -16216.409,E2 -16216.409} C_VEL
LIN {X 0,Y 298.496,Z 307.929,A -85,B 0,C 180,E1 -16219.647,E2 -16219.647} C_VEL
LIN {X 0,Y 298.427,Z 307.937,A -85,B 0,C 180,E1 -16223.6,E2 -16223.6} C_VEL
LIN {X 0,Y 298.485,Z 307.931,A -85,B 0,C 180,E1 -16226.575,E2 -16226.575} C_VEL
LIN {X 0,Y 298.415,Z 307.944,A -85,B 0,C 180,E1 -16229.641,E2 -16229.641} C_VEL
LIN {X 0,Y 298.393,Z 307.949,A -85,B 0,C 180,E1 -16232.8,E2 -16232.8} C_VEL
LIN {X 0,Y 298.417,Z 307.947,A -85,B 0,C 180,E1 -16236.07,E2 -16236.07} C_VEL
LIN {X 0,Y 298.775,Z 310.421,A -85,B 0,C 180,E1 -16239.428,E2 -16239.428} C_VEL
LIN {X 0,Y 299.253,Z 313.595,A -85,B 0,C 180,E1 -16243.278,E2 -16243.278} C_VEL
LIN {X 0,Y 299.576,Z 316.628,A -85,B 0,C 180,E1 -16246.656,E2 -16246.656} C_VEL
LIN {X 0,Y 299.498,Z 318.829,A -85,B 0,C 180,E1 -16248.925,E2 -16248.925} C_VEL
LIN {X 0,Y 299.121,Z 322.3,A -85,B 0,C 180,E1 -16252.347,E2 -16252.347} C_VEL
LIN {X 0,Y 298.77,Z 324.618,A -85,B 0,C 180,E1 -16254.524,E2 -16254.524} C_VEL
LIN {X 0,Y 299.762,Z 327.818,A -85,B 0,C 180,E1 -16254.761,E2 -16254.761} C_VEL
LIN {X 0,Y 304.637,Z 339.595,A -85,B 0,C 180,E1 -16255.86,E2 -16255.86} C_VEL
LIN {X 0,Y 309.493,Z 354.587,A -85,B 0,C 180,E1 -16257.301,E2 -16257.301} C_VEL
LIN {X 0,Y 312.7,Z 367.828,A -85,B 0,C 180,E1 -16258.656,E2 -16258.656} C_VEL
LIN {X 0,Y 314.919,Z 380.334,A -85,B 0,C 180,E1 -16260.04,E2 -16260.04} C_VEL
LIN {X 0,Y 315.477,Z 385.684,A -85,B 0,C 180,E1 -16260.653,E2 -16260.653} C_VEL
LIN {X 0,Y 312.935,Z 399.251,A -85,B 0,C 180,E1 -16262.042,E2 -16262.042} C_VEL
LIN {X 0,Y 310.093,Z 412.789,A -85,B 0,C 180,E1 -16263.771,E2 -16263.771} C_VEL
LIN {X 0,Y 307.42,Z 424.968,A -85,B 0,C 180,E1 -16265.701,E2 -16265.701} C_VEL
LIN {X 0,Y 305.418,Z 433.561,A -85,B 0,C 180,E1 -16267.329,E2 -16267.329} C_VEL
LIN {X 0,Y 303.274,Z 442.466,A -85,B 0,C 180,E1 -16269.304,E2 -16269.304} C_VEL
LIN {X 0,Y 301.259,Z 451.234,A -85,B 0,C 180,E1 -16271.643,E2 -16271.643} C_VEL
LIN {X 0,Y 299.433,Z 459.135,A -85,B 0,C 180,E1 -16274.219,E2 -16274.219} C_VEL
LIN {X 0,Y 298.119,Z 466.033,A -85,B 0,C 180,E1 -16277.058,E2 -16277.058} C_VEL
LIN {X 0,Y 297.201,Z 471.183,A -85,B 0,C 180,E1 -16279.784,E2 -16279.784} C_VEL
LIN {X 0,Y 296.812,Z 474.164,A -85,B 0,C 180,E1 -16281.832,E2 -16281.832} C_VEL
LIN {X 0,Y 296.511,Z 477.065,A -85,B 0,C 180,E1 -16284.559,E2 -16284.559} C_VEL
LIN {X 0,Y 296.475,Z 478.796,A -85,B 0,C 180,E1 -16287.282,E2 -16287.282} C_VEL
LIN {X 0,Y 296.449,Z 479.387,A -85,B 0,C 180,E1 -16289.999,E2 -16289.999} C_VEL
LIN {X 0,Y 296.476,Z 478.787,A -85,B 0,C 180,E1 -16292.717,E2 -16292.717} C_VEL
LIN {X 0,Y 296.511,Z 477.044,A -85,B 0,C 180,E1 -16295.44,E2 -16295.44} C_VEL
LIN {X 0,Y 296.811,Z 474.136,A -85,B 0,C 180,E1 -16298.167,E2 -16298.167} C_VEL
LIN {X 0,Y 297.351,Z 469.991,A -85,B 0,C 180,E1 -16300.899,E2 -16300.899} C_VEL
LIN {X 0,Y 298.418,Z 464.502,A -85,B 0,C 180,E1 -16303.621,E2 -16303.621} C_VEL
LIN {X 0,Y 299.765,Z 457.515,A -85,B 0,C 180,E1 -16306.339,E2 -16306.339} C_VEL
